(* Logix 5000 project; controller RSL5k_18_Template_noLib Emulate 5570 rev 32.11; software revision 32.02; part 13 of 16 *)
(* tags used below, declared in another part *)
   Ref_FaultCodeList : P_DescList[1];   // Tag containing List of Fault Codes (DINT) and their Descriptions (STRING)
   Inp_LastFaultCode : DINT;   // Most recent drive fault code (enumeration)
   Inp_Ready : BOOL;   // 1=Drive is ready to run
   Inp_Running : BOOL;   // 1=Drive is Running (active)
   Inp_CommandDir : BOOL;   // 1=Drive is commanded Forward, 0=Drive is commanded Reverse
   Inp_Faulted : BOOL;   // 1=Drive has Faulted (see drive display or manual)
   Inp_FwdPermOK : BOOL;   // 1=Permissives OK, drive can start Forward
   Inp_FwdNBPermOK : BOOL;   // 1=Non-Bypassable Permissives OK, drive can start Forward
   Inp_RevPermOK : BOOL;   // 1=Permissives OK, drive can start Reverse
   Inp_RevNBPermOK : BOOL;   // 1=Non-Bypassable Permissives OK, motor can start Reverse
   Inp_IntlkOK : BOOL;   // 1=Interlocks OK, drive can start/run
   Inp_NBIntlkOK : BOOL;   // 1=Non-Bypassable Interlocks OK, drive can start/run
   Inp_IntlkAvail : BOOL;   // 1 = Interlock Availibility OK
   Inp_IOFault : BOOL;   // Input Communication Status 0=OK, 1=fail
   Inp_Sim : BOOL;   // 1=Simulate working drive; 0=Start/Stop/ Monitor actual drive
   Inp_OvrdCmd : DINT;   // Override Command: 0=None, 1=Stop, 2=Start Fwd 3=Start Rev
   Cfg_HasReverse : BOOL;   // 1=Drive can be run reverse, 0=Forward only
   Cfg_HasJog : BOOL;   // 1=Drive Jog Command enabled/visible, 0=Drive Jog Command not allowed
   Cfg_AllowLocal : BOOL;   // 1=Allow Local Start/Stop without alarm, 0=Start/Stop from HMI/prog only
   Cfg_HasRunFdbk : BOOL;   // 1=Drive provides feedback signal on Inp_Running when running
   Cfg_UseRunFdbk : BOOL;   // 1=Drive run feedback should be used for failure checking
   Cfg_HasSpeedFdbk : BOOL;   // 1=Drive provides speed feedback on Inp_SpeedFdbk
   Cfg_HasOutDatalink : BOOL;   // 1=A signal is connected to Out_Datalink
   Cfg_SetTrack : BOOL;   // 1=Settings track for unselected sources, 0=no tracking
   Cfg_SetTrackOvrdHand : BOOL;   // 1=Prog/Oper/Ext Settings track Override/Hand
   Cfg_OperStopPrio : BOOL;   // 1=OCmd_Stop any time, 0=OCmd_Stop only when Oper selected
   Cfg_ExtStopPrio : BOOL;   // 1=XCmd_Stop any time, 0=XCmd_Stop only when Ext selected
   Cfg_OCmdResets : BOOL;   // 1=New drive OCmd resets shed latches and cleared alarms, 0=OCmdReset req'd.
   Cfg_ShedOnFailToStart : BOOL;   // 1=Stop Motor and Alarm on Fail to Start; 0=Alarm only on Fail to Start
   Cfg_ShedOnIOFault : BOOL;   // 1=Stop Motor and Alarm on I/O Fault; 0=Alarm only on I/O Fault
   Cfg_MinSpdRef : REAL;   // Minimum Speed Reference in EU (for limiting)
   Cfg_MaxSpdRef : REAL;   // Maximum Speed Reference in EU (for limiting)
   Cfg_SpeedRefRawMin : REAL;   // Speed Reference Minimum in Drive (raw) Units (for scaling)
   Cfg_SpeedRefRawMax : REAL;   // Speed Reference Maximum in Drive (raw) Units (for scaling)
   Cfg_SpeedRefEUMin : REAL;   // Speed Reference Minimum in Engineering Units (for scaling)
   Cfg_SpeedRefEUMax : REAL;   // Speed Reference Maximum in Engineering Units (for scaling)
   Cfg_OutDatalinkRawMin : REAL;   // Output Datalink Minimum in Drive (raw) Units (for scaling)
   Cfg_OutDatalinkRawMax : REAL;   // Output Datalink Maximum in Drive (raw) Units (for scaling)
   Cfg_OutDatalinkEUMin : REAL;   // Output Datalink Minimum in Engineering Units (for scaling)
   Cfg_OutDatalinkEUMax : REAL;   // Output Datalink Maximum in Engineering Units (for scaling)
   PSet_SpeedRef : REAL;   // Program Setting of Speed Reference (EU)
   PSet_OutDatalink : REAL;   // Program Setting of Output Datalink (EU)
   XSet_SpeedRef : REAL;   // External Setting of Speed Reference (EU)
   XSet_OutDatalink : REAL;   // External Setting of Output Datalink (EU)
   PCmd_StartFwd : BOOL;   // Program Command to Start Drive Forward
   PCmd_StartRev : BOOL;   // Program Command to Start Drive Reverse
   PCmd_Stop : BOOL;   // Program Command to Stop Drive
   PCmd_Reset : BOOL;   // Program Command to Reset drive fault and all Alarms requiring Reset
   XCmd_StartFwd : BOOL;   // External Command to Start Drive Forward
   XCmd_StartRev : BOOL;   // External Command to Start Drive Reverse
   XCmd_Stop : BOOL;   // External Command to Stop Drive
   XCmd_JogFwd : BOOL;   // External Command to Jog Drive Forward
   XCmd_JogRev : BOOL;   // External Command to Jog Drive Reverse
   Out_SpeedRef : REAL;   // Drive Speed Reference in Drive Units (typ. 0-32767 = 0 to max freq.)
   Out_Datalink : REAL;   // Auxiliary Signal (datalink) Output in Drive (raw) Units
   Out_Run : BOOL;   // 1=Start/Run Drive, 0=Stop Drive (for held starter type)
   Out_Stop : BOOL;   // 1=Stop Drive, 0=drive left in current state
   Out_Start : BOOL;   // 1=Start Drive, 0=drive left in current state
   Out_Jog : BOOL;   // 1=Jog drive at Jog Speed, -->0=stop jogging
   Out_ClearFault : BOOL;   // 1=Attempt to clear Drive Fault
   Out_Fwd : BOOL;   // 1=Set drive direction to Forward
   Out_Rev : BOOL;   // 1=Set drive direction to Reverse
   Out_Horn : BOOL;   // 1=Sound audible prior to commanded motor start
   Val_SpeedRef : REAL;   // Speed Reference (target) to drive
   Val_OutDatalink : REAL;   // Output Datalink value to drive
   Val_LastFaultCode : DINT;   // Most recent drive fault code (enumeration)
   Val_Cmd : DINT;   // Device Command 0=None, 1=Stop, 2=StartFwd 3=StartRev 4=JogFwd 5=JogRev
   Sts_Stopped : BOOL;   // 1=Drive requested to stop and is confirmed stopped
   Sts_StartingFwd : BOOL;   // 1=Drive requested to run forward and awaiting run feedback
   Sts_StartingRev : BOOL;   // 1=Drive requested to run reverse and awaiting run feedback
   Sts_RunningFwd : BOOL;   // 1=Drive requested to run and is confirmed running forward
   Sts_RunningRev : BOOL;   // 1=Drive requested to run and is confirmed running reverse
   Sts_StoppingFwd : BOOL;   // 1=Drive running forward requested to stop and awaiting stopped feedback
   Sts_StoppingRev : BOOL;   // 1=Drive running reverse requested to stop and awaiting stopped feedback
   Sts_JoggingFwd : BOOL;   // 1=Drive requested to Jog Forward
   Sts_JoggingRev : BOOL;   // 1=Drive requested to Jog Reverse
   Sts_Horn : BOOL;   // 1=Motor Horn Active
   Sts_CommandDir : BOOL;   // 1=Drive commanded to Forward, 0=Reverse
   Sts_ActualDir : BOOL;   // 1=Drive Actual direction is Forward, 0=Reverse
   Sts_SpeedLimited : BOOL;   // 1=Speed Reference Setting exceeds configured Max/Min limit
   Sts_Available : BOOL;   // 1=Drive available for control by automation (Prog)
   Sts_BypActive : BOOL;   // 1=Bypassing Active (Bypassed or Maintenance)
   Sts_NotRdy : BOOL;   // 1=Device Not Ready, see detail bits for reason
   Nrdy_CfgErr : BOOL;   // 1=Device Not Ready: Configuration Error
   Nrdy_DriveNR : BOOL;   // 1=Device Note Ready: Drive Not Ready
   Nrdy_Fail : BOOL;   // 1=Device Not Ready: Device Failure (Shed Requires Reset)
   Nrdy_Intlk : BOOL;   // 1=Device Not Ready: Interlock Not OK
   Nrdy_IOFault : BOOL;   // 1=Device Not Ready: I/O Fault (Shed Requires Reset)
   Nrdy_OoS : BOOL;   // 1=Device Not Ready: Device is Out of Service
   Nrdy_Perm : BOOL;   // 1=Device Not Ready: Permissive Not OK
   Nrdy_PrioStop : BOOL;   // 1=Device Not Ready: Oper/Ext Priority Stop Requires Reset
   Nrdy_Trip : BOOL;   // 1=Device not Ready: Deivce Tripped (Drive Fault)
   Sts_AlmInh : BOOL;   // 1=An Alarm is Shelved, Disabled or Suppressed, display icon
   Err_RefEU : BOOL;   // 1=Error in Config: Speed Ref EU Min = Max
   Err_OutDLEU : BOOL;   // 1=Error in Config: Output Datalink EU Min = Max
   Sts_Hand : ALIAS FOR CmdSrc.Sts_Hand;
   Sts_OoS : ALIAS FOR CmdSrc.Sts_OoS;
   Sts_Maint : ALIAS FOR CmdSrc.Sts_Maint;
   Sts_Ovrd : ALIAS FOR CmdSrc.Sts_Ovrd;
   Sts_Prog : ALIAS FOR CmdSrc.Sts_Prog;
   Sts_Oper : ALIAS FOR CmdSrc.Sts_Oper;
   Sts_FailToStart : ALIAS FOR FailToStart.Inp;   // 1=Drive Failed to Start (One-Shot)
   Sts_FailToStop : ALIAS FOR FailToStop.Inp;   // 1=Drive Failed to Stop
   Sts_IntlkTrip : ALIAS FOR IntlkTrip.Inp;   // 1=Drive was stopped by an Interlock NOT OK (One-Shot)
   Sts_DriveFault : ALIAS FOR DriveFault.Inp;   // 1=Drive Fault (see drive display or manual)
   Sts_IOFault : ALIAS FOR IOFault.Inp;   // I/O Comm Fault Status (0=OK, 1=Bad)
   P_VSD : BOOL;   // Unique Parameter Name for auto - discovery
   CmdSrc : P_CmdSrc;   // Drive Mode Selection
   IOFault : P_Alarm;   // I/O Fault Alarm
   IntlkTrip : P_Alarm;   // Interlock Trip Alarm
   FailToStop : P_Alarm;   // Drive Failed to Stop Alarm
   FailToStart : P_Alarm;   // Drive Failed to Start Alarm
   Wrk_Run : BOOL;   // 1=Drive should be "running", 0=should be "stopped"
   Wrk_StartRetrigT : TIMER;   // Time to pulse start output on start command retrigger (Maint)
   Wrk_StopRetrigT : TIMER;   // Time to pulse stop output on stop command retrigger (Maint)
   Wrk_RunFdbk : BOOL;   // Run Feedback based on mode, simulation, etc. 1=running
   DriveFault : P_Alarm;   // Drive Faulted Alarm
   Wrk_SpeedRef : REAL;   // Working copy of Speed Reference (for limiting)
   Wrk_Rev : BOOL;   // Working (internal) Direction 1=Reverse 0=Forward (default)
   Wrk_Jog : BOOL;   // 1=Jog Drive, 0=Drive not jogging
   Wrk_ResetT : TIMER;   // Reset Output Pulse Timer
   Wrk_OutDatalink : REAL;   // Selected Output Datalink setting
   Wrk_StopT : TIMER;   // Stop Check Timer (for Fail to Stop)
   Wrk_StartT : TIMER;   // Start Check Timer (for Fail to Start)
   Wrk_Cmd : DINT;   // Buffer for building Val_Cmd
   Wrk_Retrigger : BOOL;   // Maint Start issued while running or Stop while stopped
   Wrk_JogT : TIMER;   // Jog Timer
   Wrk_FaultDescFSC : CONTROL;   // FSC control for Fault Code List search
   Val_FaultDesc : STRING_40;   // Description of Drive Fault (given LastFaultCode)
   Wrk_NotRdyONS : BOOL;   // Assert Stop on One-Shot of Sts_NotRdy
   Wrk_NotRdy : BOOL;   // Device Not Ready conditions excluding shed latches
   Wrk_StartInhT : TIMER;   // Local Start Inhibit Timer
   Wrk_StopInhT : TIMER;   // Local Stop Inhibit Timer
   Wrk_Hand : BOOL;   // Perform Hand Mode alignment with actual device state
   Wrk_StartHornT : TIMER;   // Timer for audible alert or start
   Wrk_StartHorn : BOOL;   // 1=Sound audible prior to commanded motor start
   Wrk_RevPermOK : BOOL;   // Reverse Permissives and NB Permissive OK
   Wrk_FwdPermOK : BOOL;   // Forward Permissives and NB Permissive OK
   OCmd_JogRev : BOOL;   // Operator Command to Jog Drive Reverse (not cleared by instruction!)
   OCmd_JogFwd : BOOL;   // Operator Command to Jog Drive Forward (not cleared by instruction!)
   OCmd_Stop : BOOL;   // Operator Command to Stop Drive
   OCmd_StartRev : BOOL;   // Operator Command to Start Drive Reverse
   OCmd_StartFwd : BOOL;   // Operator Command to Start Drive Forward
   OSet_OutDatalink : REAL;   // Operator Setting of Output Datalink (EU)
   OSet_SpeedRef : REAL;   // Operator Setting of Speed Reference (EU)
   ORdy_JogRev : BOOL;   // 1=Ready for OCmd_JogRev (enabled HMI button)
   ORdy_JogFwd : BOOL;   // 1=Ready for OCmd_JogFwd (enables HMI button)
   ORdy_Stop : BOOL;   // 1=Ready for OCmd_Stop (enables HMI button)
   ORdy_StartRev : BOOL;   // 1=Ready for OCmd_StartRev (enables HMI button)
   ORdy_StartFwd : BOOL;   // 1=Ready for OCmd_StartFwd (enables HMI button)
   Wrk_ExtHas1 : BOOL;   // External has Commands
   Wrk_ProgHas1 : BOOL;   // Program has Commands
   Wrk_OperHas1 : BOOL;   // Operator has Commands
(* P_VSD, continued *)

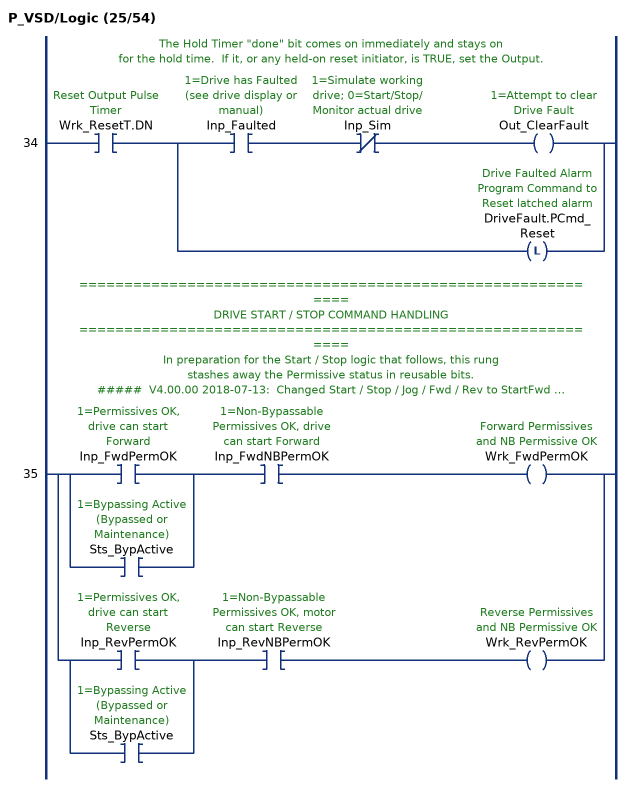
   [picture p277: P_VSD/Logic rungs 34-35]
   // The Hold Timer "done" bit comes on immediately and stays on
   // for the hold time.  If it, or any held-on reset initiator, is TRUE, set the Output.
   34: XIC(Wrk_ResetT.DN)[XIC(Inp_Faulted) XIO(Inp_Sim) OTE(Out_ClearFault) ,OTL(DriveFault.PCmd_Reset) ];
   // ============================================================
   // DRIVE START / STOP COMMAND HANDLING
   // ============================================================
   // In preparation for the Start / Stop logic that follows, this rung
   // stashes away the Permissive status in reusable bits.
   // #####  V4.00.00 2018-07-13:  Changed Start / Stop / Jog / Fwd / Rev to StartFwd / StartRev / Stop / JogFwd / JogRev  #####
   35: [[XIC(Inp_FwdPermOK) ,XIC(Sts_BypActive) ] XIC(Inp_FwdNBPermOK) OTE(Wrk_FwdPermOK) ,[XIC(Inp_RevPermOK) ,XIC(Sts_BypActive) ] XIC(Inp_RevNBPermOK) OTE(Wrk_RevPermOK) ];
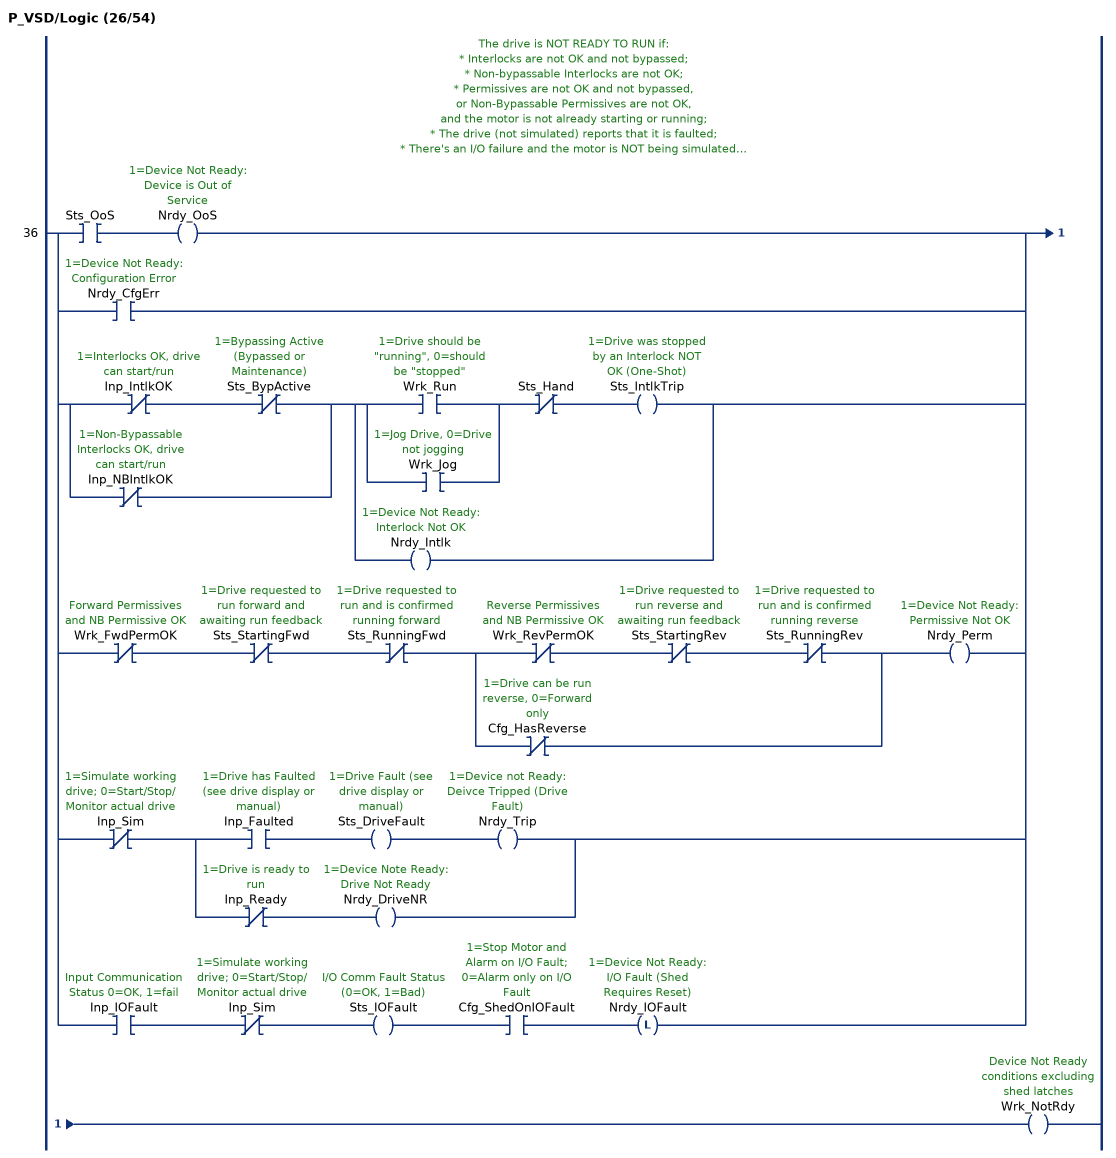
   // The drive is NOT READY TO RUN if:
   // * Interlocks are not OK and not bypassed;
   // * Non-bypassable Interlocks are not OK;
   // * Permissives are not OK and not bypassed,
   // or Non-Bypassable Permissives are not OK,
   // and the motor is not already starting or running;
   // * The drive (not simulated) reports that it is faulted;
   // * There's an I/O failure and the motor is NOT being simulated;
   // * The motor has a Fail to Start that has not been reset;
   // * The drive is disabled (by Maintenance);
   // * This instruction instance has a configuration error.
   // #####  V4.00.00  2018-07-13:  Disable/Enable replaced by P_CmdSrc Out of Service (OoS).  #####
   // #####  V4.00.00  2018-07-13:  Replaced start / stop / fwd / rev with start fwd / start rev / stop  #####
   36: [XIC(Sts_OoS) OTE(Nrdy_OoS) ,XIC(Nrdy_CfgErr) ,[XIO(Inp_IntlkOK) XIO(Sts_BypActive) ,XIO(Inp_NBIntlkOK) ] [[XIC(Wrk_Run) ,XIC(Wrk_Jog) ] XIO(Sts_Hand) OTE(Sts_IntlkTrip) ,OTE(Nrdy_Intlk) ] ,XIO(Wrk_FwdPermOK) XIO(Sts_StartingFwd) XIO(Sts_RunningFwd) [XIO(Wrk_RevPermOK) XIO(Sts_StartingRev) XIO(Sts_RunningRev) ,XIO(Cfg_HasReverse) ] OTE(Nrdy_Perm) ,XIO(Inp_Sim) [XIC(Inp_Faulted) OTE(Sts_DriveFault) OTE(Nrdy_Trip) ,XIO(Inp_Ready) OTE(Nrdy_DriveNR) ] ,XIC(Inp_IOFault) XIO(Inp_Sim) OTE(Sts_IOFault) XIC(Cfg_ShedOnIOFault) OTL(Nrdy_IOFault) ]OTE(Wrk_NotRdy);
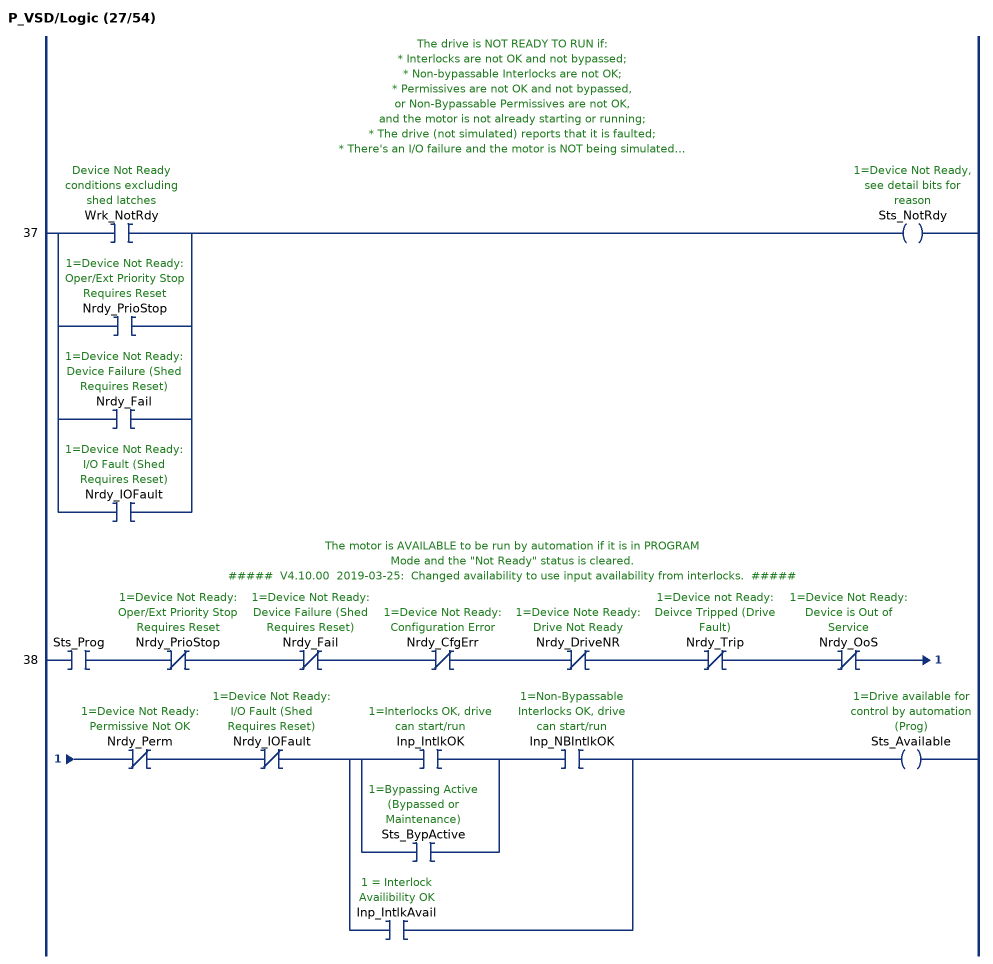
   // The drive is NOT READY TO RUN if:
   // * Interlocks are not OK and not bypassed;
   // * Non-bypassable Interlocks are not OK;
   // * Permissives are not OK and not bypassed,
   // or Non-Bypassable Permissives are not OK,
   // and the motor is not already starting or running;
   // * The drive (not simulated) reports that it is faulted;
   // * There's an I/O failure and the motor is NOT being simulated;
   // * The motor has a Fail to Start that has not been reset;
   // * The drive is disabled (by Maintenance);
   // * This instruction instance has a configuration error.
   37: [XIC(Wrk_NotRdy) ,XIC(Nrdy_PrioStop) ,XIC(Nrdy_Fail) ,XIC(Nrdy_IOFault) ]OTE(Sts_NotRdy);
   // The motor is AVAILABLE to be run by automation if it is in PROGRAM
   // Mode and the "Not Ready" status is cleared.
   // #####  V4.10.00  2019-03-25:  Changed availability to use input availability from interlocks.  #####
   38: XIC(Sts_Prog)XIO(Nrdy_PrioStop)XIO(Nrdy_Fail)XIO(Nrdy_CfgErr)XIO(Nrdy_DriveNR)XIO(Nrdy_Trip)XIO(Nrdy_OoS)XIO(Nrdy_Perm)XIO(Nrdy_IOFault)[[XIC(Inp_IntlkOK) ,XIC(Sts_BypActive) ] XIC(Inp_NBIntlkOK) ,XIC(Inp_IntlkAvail) ]OTE(Sts_Available);
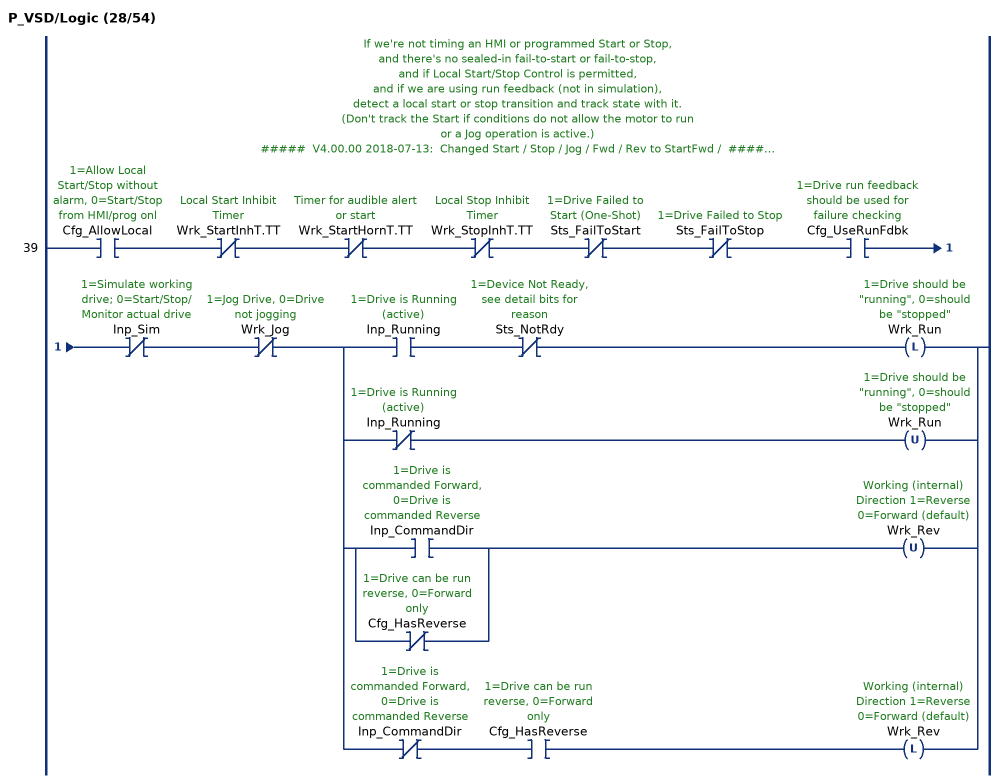
   // If we're not timing an HMI or programmed Start or Stop,
   // and there's no sealed-in fail-to-start or fail-to-stop,
   // and if Local Start/Stop Control is permitted,
   // and if we are using run feedback (not in simulation),
   // detect a local start or stop transition and track state with it.
   // (Don't track the Start if conditions do not allow the motor to run
   // or a Jog operation is active.)
   // #####  V4.00.00 2018-07-13:  Changed Start / Stop / Jog / Fwd / Rev to StartFwd /  #####
   // #####  StartRev / Stop / JogFwd / JogRev.  Deleted Cfg_PCmdClear.  #####
   // ##### V4.00.02  2018-10-30:  Corrected handling Allow Local when horn is enabled.  #####
   39: XIC(Cfg_AllowLocal)XIO(Wrk_StartInhT.TT)XIO(Wrk_StartHornT.TT)XIO(Wrk_StopInhT.TT)XIO(Sts_FailToStart)XIO(Sts_FailToStop)XIC(Cfg_UseRunFdbk)XIO(Inp_Sim)XIO(Wrk_Jog)[XIC(Inp_Running) XIO(Sts_NotRdy) OTL(Wrk_Run) ,XIO(Inp_Running) OTU(Wrk_Run) ,[XIC(Inp_CommandDir) ,XIO(Cfg_HasReverse) ] OTU(Wrk_Rev) ,XIO(Inp_CommandDir) XIC(Cfg_HasReverse) OTL(Wrk_Rev) ];
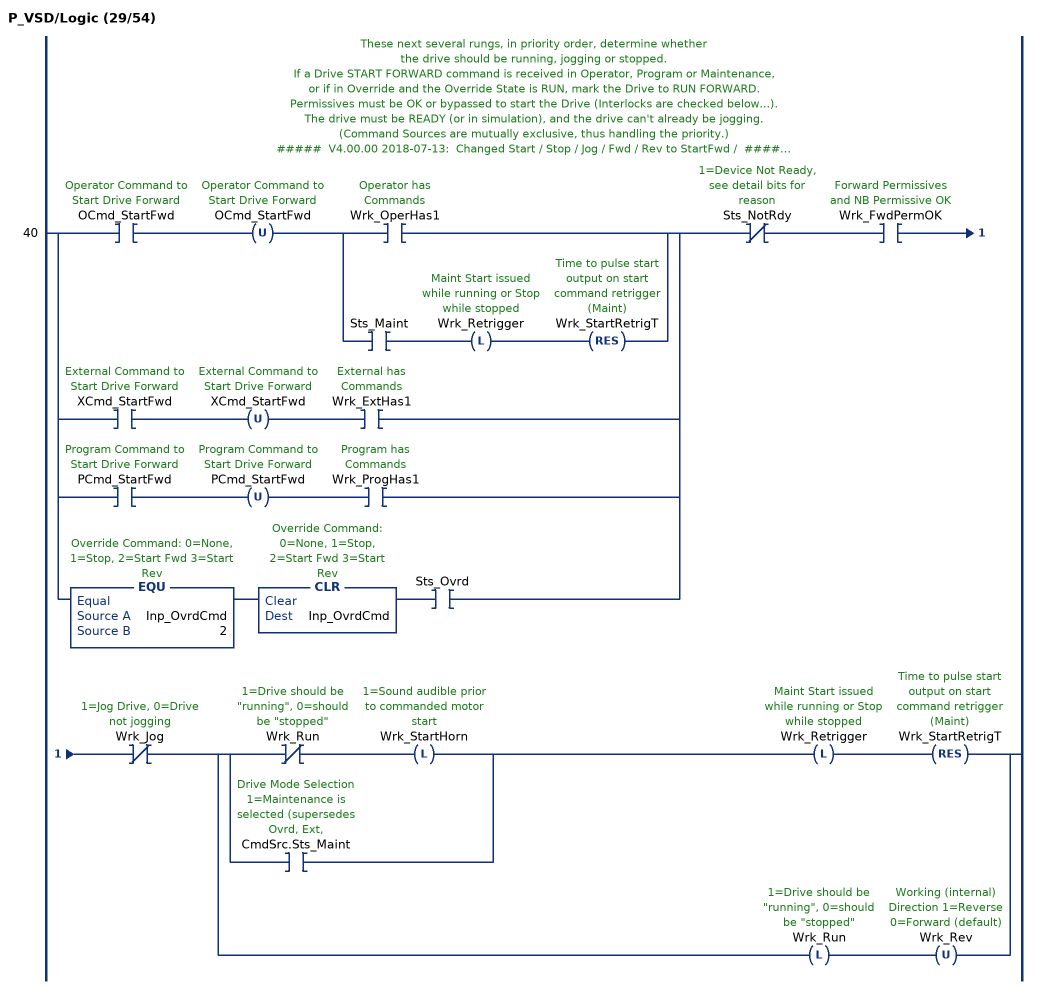
   // These next several rungs, in priority order, determine whether
   // the drive should be running, jogging or stopped.
   // If a Drive START FORWARD command is received in Operator, Program or Maintenance,
   // or if in Override and the Override State is RUN, mark the Drive to RUN FORWARD.
   // Permissives must be OK or bypassed to start the Drive (Interlocks are checked below...).
   // The drive must be READY (or in simulation), and the drive can't already be jogging.
   // (Command Sources are mutually exclusive, thus handling the priority.)
   // #####  V4.00.00 2018-07-13:  Changed Start / Stop / Jog / Fwd / Rev to StartFwd /  #####
   // #####  StartRev / Stop / JogFwd / JogRev.  Deleted Cfg_PCmdClear.  #####
   // #####  Added audible alert prior to commanded start.  #####
   // #####  Changed P_Mode to P_CmdSrc. Added External Command Source and Commands.  #####
   40: [XIC(OCmd_StartFwd) OTU(OCmd_StartFwd) [XIC(Wrk_OperHas1) ,XIC(Sts_Maint) OTL(Wrk_Retrigger) RES(Wrk_StartRetrigT) ] ,XIC(XCmd_StartFwd) OTU(XCmd_StartFwd) XIC(Wrk_ExtHas1) ,XIC(PCmd_StartFwd) OTU(PCmd_StartFwd) XIC(Wrk_ProgHas1) ,EQU(Inp_OvrdCmd,2) CLR(Inp_OvrdCmd) XIC(Sts_Ovrd) ]XIO(Sts_NotRdy)XIC(Wrk_FwdPermOK)XIO(Wrk_Jog)[[XIO(Wrk_Run) OTL(Wrk_StartHorn) ,XIC(CmdSrc.Sts_Maint) ] OTL(Wrk_Retrigger) RES(Wrk_StartRetrigT) ,OTL(Wrk_Run) OTU(Wrk_Rev) ];
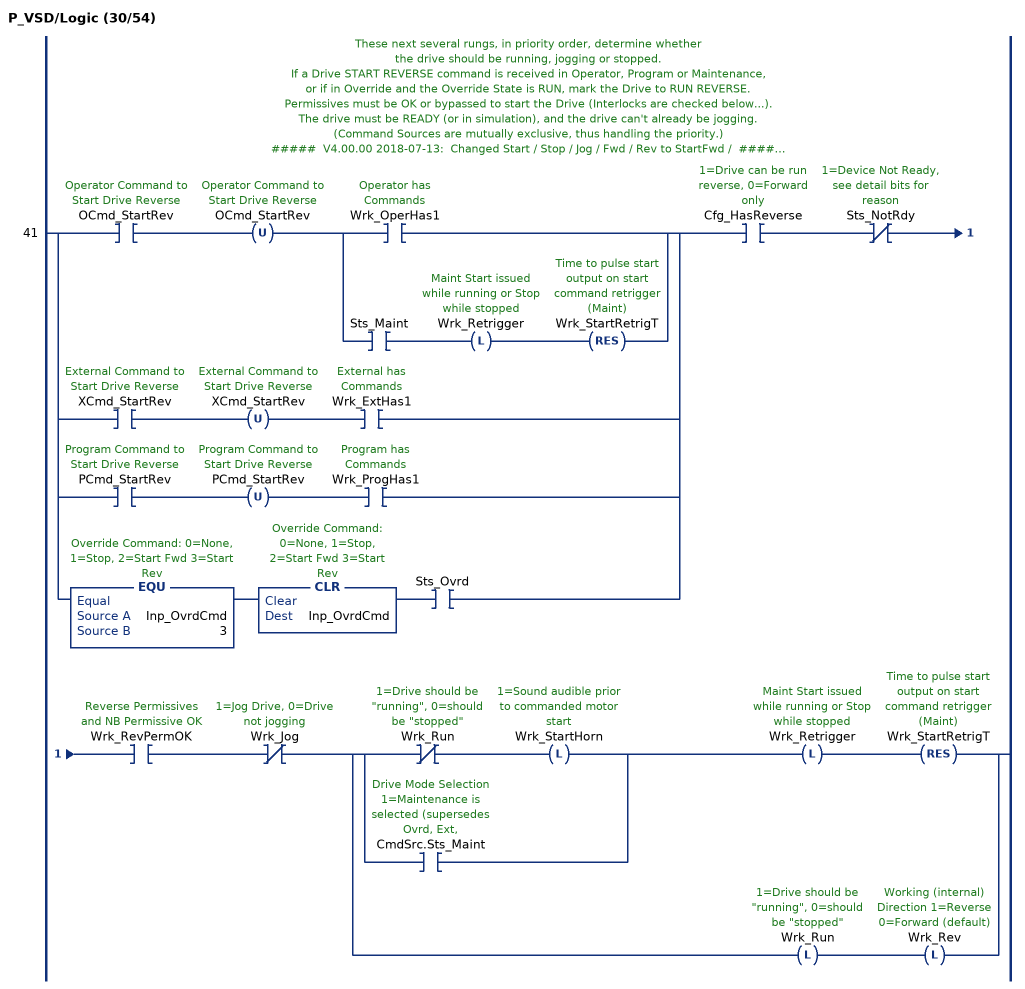
   // These next several rungs, in priority order, determine whether
   // the drive should be running, jogging or stopped.
   // If a Drive START REVERSE command is received in Operator, Program or Maintenance,
   // or if in Override and the Override State is RUN, mark the Drive to RUN REVERSE.
   // Permissives must be OK or bypassed to start the Drive (Interlocks are checked below...).
   // The drive must be READY (or in simulation), and the drive can't already be jogging.
   // (Command Sources are mutually exclusive, thus handling the priority.)
   // #####  V4.00.00 2018-07-13:  Changed Start / Stop / Jog / Fwd / Rev to StartFwd /  #####
   // #####  StartRev / Stop / JogFwd / JogRev.  Deleted Cfg_PCmdClear.  #####
   // #####  Added audible alert prior to commanded start.  #####
   // #####  Changed P_Mode to P_CmdSrc. Added External Command Source and Commands.  #####
   41: [XIC(OCmd_StartRev) OTU(OCmd_StartRev) [XIC(Wrk_OperHas1) ,XIC(Sts_Maint) OTL(Wrk_Retrigger) RES(Wrk_StartRetrigT) ] ,XIC(XCmd_StartRev) OTU(XCmd_StartRev) XIC(Wrk_ExtHas1) ,XIC(PCmd_StartRev) OTU(PCmd_StartRev) XIC(Wrk_ProgHas1) ,EQU(Inp_OvrdCmd,3) CLR(Inp_OvrdCmd) XIC(Sts_Ovrd) ]XIC(Cfg_HasReverse)XIO(Sts_NotRdy)XIC(Wrk_RevPermOK)XIO(Wrk_Jog)[[XIO(Wrk_Run) OTL(Wrk_StartHorn) ,XIC(CmdSrc.Sts_Maint) ] OTL(Wrk_Retrigger) RES(Wrk_StartRetrigT) ,OTL(Wrk_Run) OTL(Wrk_Rev) ];
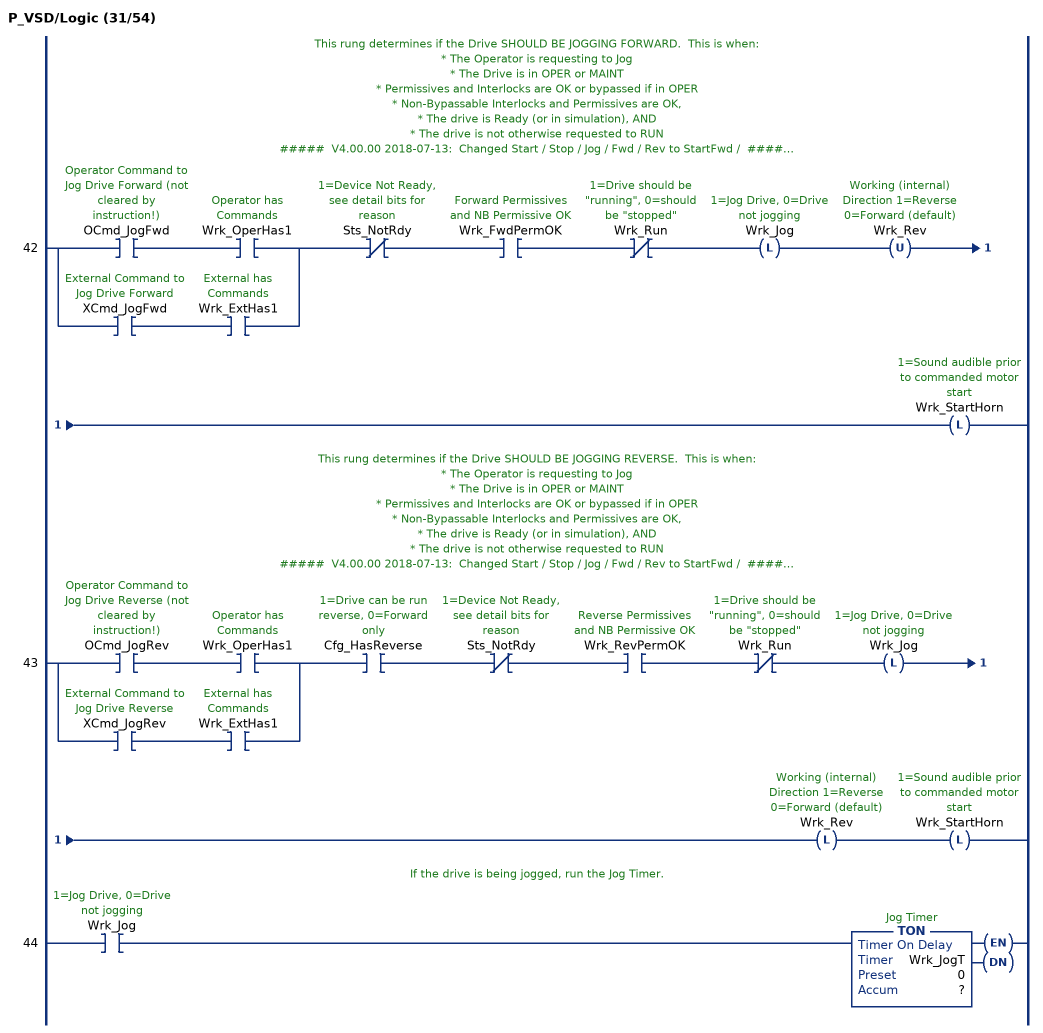
   // This rung determines if the Drive SHOULD BE JOGGING FORWARD.  This is when:
   // * The Operator is requesting to Jog
   // * The Drive is in OPER or MAINT
   // * Permissives and Interlocks are OK or bypassed if in OPER
   // * Non-Bypassable Interlocks and Permissives are OK,
   // * The drive is Ready (or in simulation), AND
   // * The drive is not otherwise requested to RUN
   // #####  V4.00.00 2018-07-13:  Changed Start / Stop / Jog / Fwd / Rev to StartFwd /  #####
   // #####  StartRev / Stop / JogFwd / JogRev.  Deleted Cfg_PCmdClear.  #####
   // #####  Changed P_Mode to P_CmdSrc. Added External Command Source and Commands.  #####
   42: [XIC(OCmd_JogFwd) XIC(Wrk_OperHas1) ,XIC(XCmd_JogFwd) XIC(Wrk_ExtHas1) ]XIO(Sts_NotRdy)XIC(Wrk_FwdPermOK)XIO(Wrk_Run)OTL(Wrk_Jog)OTU(Wrk_Rev)OTL(Wrk_StartHorn);
   // This rung determines if the Drive SHOULD BE JOGGING REVERSE.  This is when:
   // * The Operator is requesting to Jog
   // * The Drive is in OPER or MAINT
   // * Permissives and Interlocks are OK or bypassed if in OPER
   // * Non-Bypassable Interlocks and Permissives are OK,
   // * The drive is Ready (or in simulation), AND
   // * The drive is not otherwise requested to RUN
   // #####  V4.00.00 2018-07-13:  Changed Start / Stop / Jog / Fwd / Rev to StartFwd /  #####
   // #####  StartRev / Stop / JogFwd / JogRev.  Deleted Cfg_PCmdClear.  #####
   // #####  Changed P_Mode to P_CmdSrc. Added External Command Source and Commands.  #####
   43: [XIC(OCmd_JogRev) XIC(Wrk_OperHas1) ,XIC(XCmd_JogRev) XIC(Wrk_ExtHas1) ]XIC(Cfg_HasReverse)XIO(Sts_NotRdy)XIC(Wrk_RevPermOK)XIO(Wrk_Run)OTL(Wrk_Jog)OTL(Wrk_Rev)OTL(Wrk_StartHorn);
   // If the drive is being jogged, run the Jog Timer.
   44: XIC(Wrk_Jog)TON(Wrk_JogT,?,?);
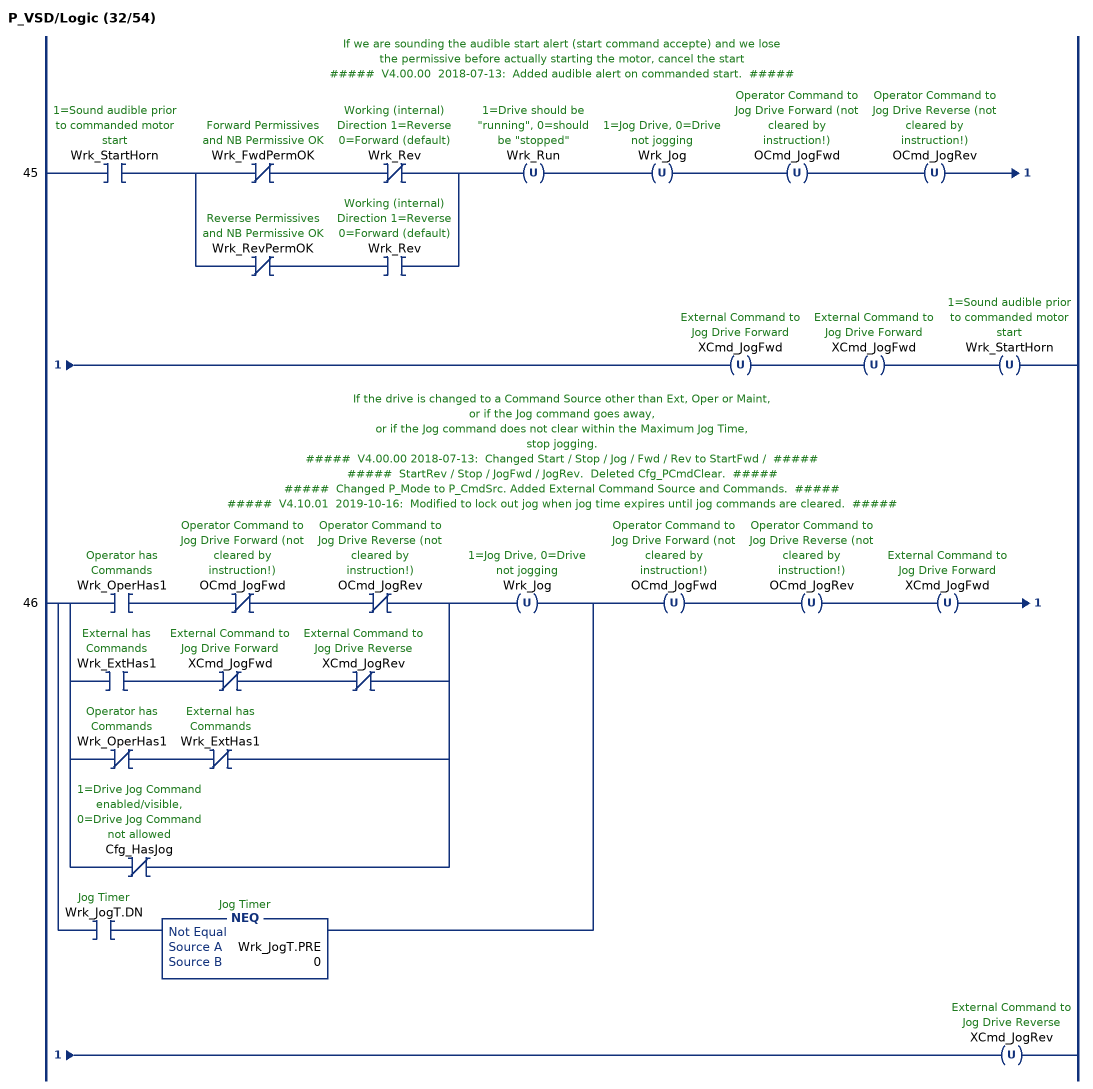
   // If we are sounding the audible start alert (start command accepte) and we lose
   // the permissive before actually starting the motor, cancel the start
   // #####  V4.00.00  2018-07-13:  Added audible alert on commanded start.  #####
   45: XIC(Wrk_StartHorn)[XIO(Wrk_FwdPermOK) XIO(Wrk_Rev) ,XIO(Wrk_RevPermOK) XIC(Wrk_Rev) ]OTU(Wrk_Run)OTU(Wrk_Jog)OTU(OCmd_JogFwd)OTU(OCmd_JogRev)OTU(XCmd_JogFwd)OTU(XCmd_JogFwd)OTU(Wrk_StartHorn);
   // If the drive is changed to a Command Source other than Ext, Oper or Maint,
   // or if the Jog command goes away,
   // or if the Jog command does not clear within the Maximum Jog Time,
   // stop jogging.
   // #####  V4.00.00 2018-07-13:  Changed Start / Stop / Jog / Fwd / Rev to StartFwd /  #####
   // #####  StartRev / Stop / JogFwd / JogRev.  Deleted Cfg_PCmdClear.  #####
   // #####  Changed P_Mode to P_CmdSrc. Added External Command Source and Commands.  #####
   // #####  V4.10.01  2019-10-16:  Modified to lock out jog when jog time expires until jog commands are cleared.  #####
   46: [[XIC(Wrk_OperHas1) XIO(OCmd_JogFwd) XIO(OCmd_JogRev) ,XIC(Wrk_ExtHas1) XIO(XCmd_JogFwd) XIO(XCmd_JogRev) ,XIO(Wrk_OperHas1) XIO(Wrk_ExtHas1) ,XIO(Cfg_HasJog) ] OTU(Wrk_Jog) ,XIC(Wrk_JogT.DN) NEQ(Wrk_JogT.PRE,0) ]OTU(OCmd_JogFwd)OTU(OCmd_JogRev)OTU(XCmd_JogFwd)OTU(XCmd_JogRev);
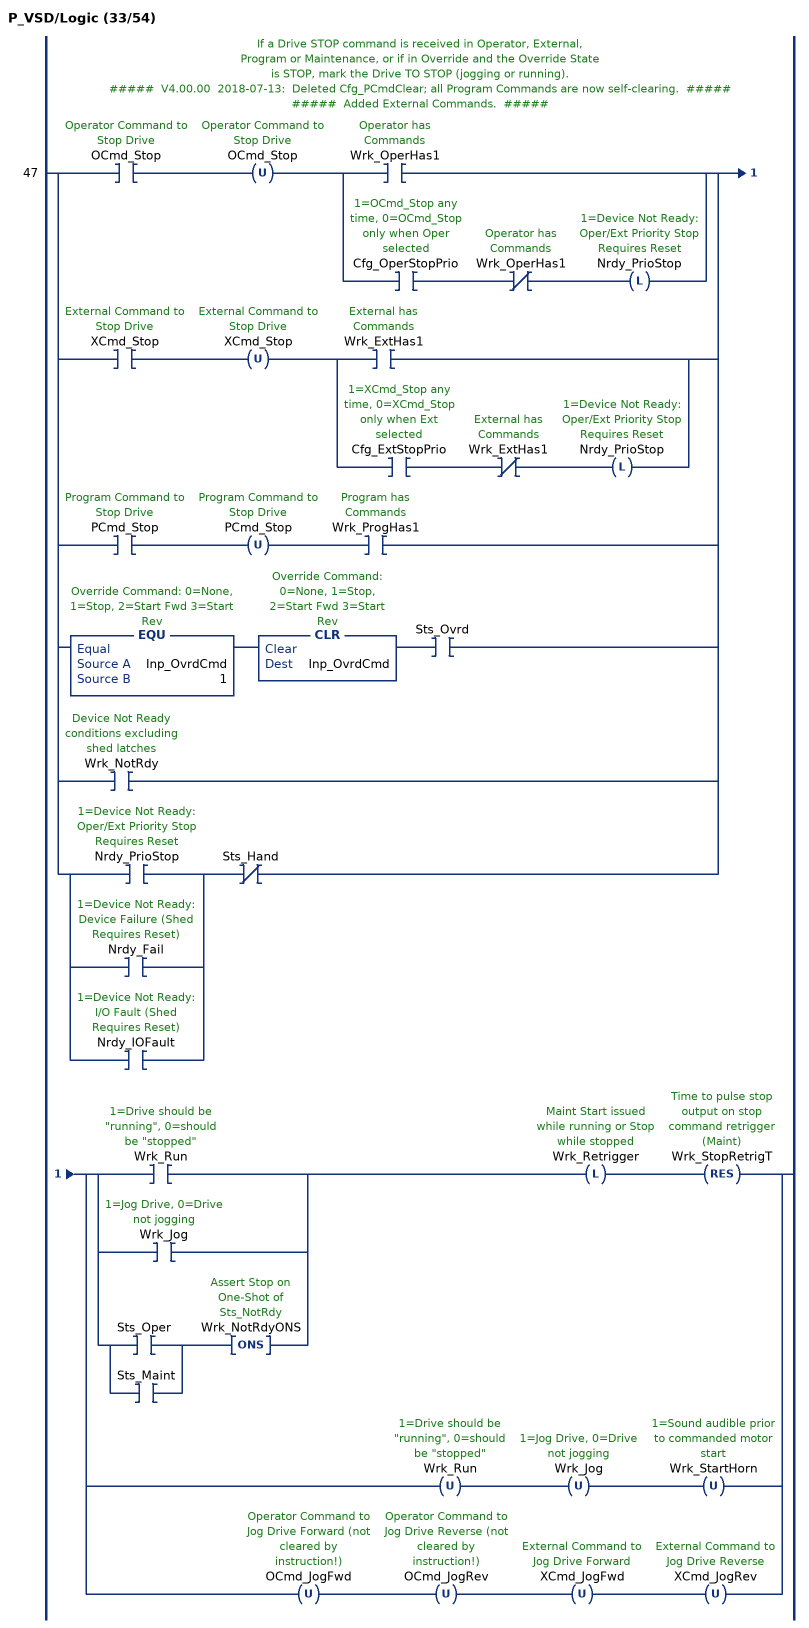
   // If a Drive STOP command is received in Operator, External,
   // Program or Maintenance, or if in Override and the Override State
   // is STOP, mark the Drive TO STOP (jogging or running).
   // #####  V4.00.00  2018-07-13:  Deleted Cfg_PCmdClear; all Program Commands are now self-clearing.  #####
   // #####  Added External Commands.  #####
   47: [XIC(OCmd_Stop) OTU(OCmd_Stop) [XIC(Wrk_OperHas1) ,XIC(Cfg_OperStopPrio) XIO(Wrk_OperHas1) OTL(Nrdy_PrioStop) ] ,XIC(XCmd_Stop) OTU(XCmd_Stop) [XIC(Wrk_ExtHas1) ,XIC(Cfg_ExtStopPrio) XIO(Wrk_ExtHas1) OTL(Nrdy_PrioStop) ] ,XIC(PCmd_Stop) OTU(PCmd_Stop) XIC(Wrk_ProgHas1) ,EQU(Inp_OvrdCmd,1) CLR(Inp_OvrdCmd) XIC(Sts_Ovrd) ,XIC(Wrk_NotRdy) ,[XIC(Nrdy_PrioStop) ,XIC(Nrdy_Fail) ,XIC(Nrdy_IOFault) ] XIO(Sts_Hand) ][[XIC(Wrk_Run) ,XIC(Wrk_Jog) ,[XIC(Sts_Oper) ,XIC(Sts_Maint) ] ONS(Wrk_NotRdyONS) ] OTL(Wrk_Retrigger) RES(Wrk_StopRetrigT) ,OTU(Wrk_Run) OTU(Wrk_Jog) OTU(Wrk_StartHorn) ,OTU(OCmd_JogFwd) OTU(OCmd_JogRev) OTU(XCmd_JogFwd) OTU(XCmd_JogRev) ];
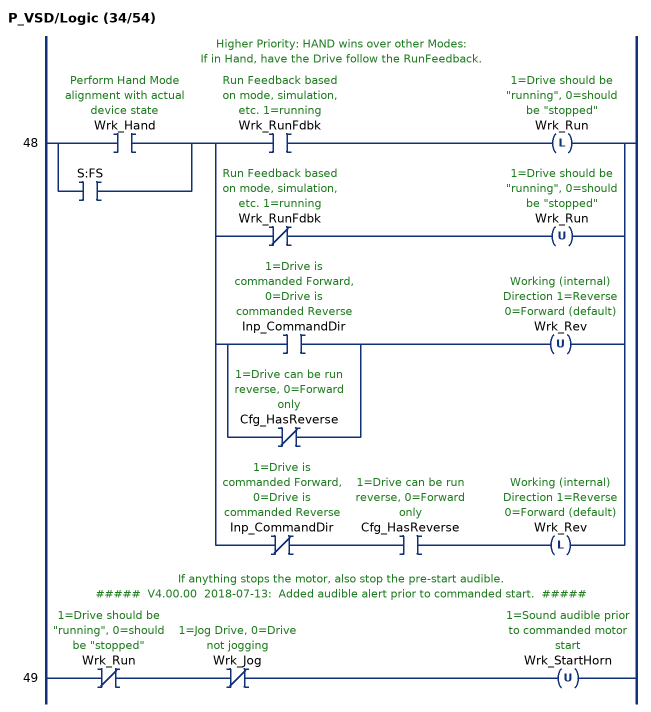
   // Higher Priority: HAND wins over other Modes:
   // If in Hand, have the Drive follow the RunFeedback.
   48: [XIC(Wrk_Hand) ,XIC(S:FS) ][XIC(Wrk_RunFdbk) OTL(Wrk_Run) ,XIO(Wrk_RunFdbk) OTU(Wrk_Run) ,[XIC(Inp_CommandDir) ,XIO(Cfg_HasReverse) ] OTU(Wrk_Rev) ,XIO(Inp_CommandDir) XIC(Cfg_HasReverse) OTL(Wrk_Rev) ];
   // If anything stops the motor, also stop the pre-start audible.
   // #####  V4.00.00  2018-07-13:  Added audible alert prior to commanded start.  #####
   49: XIO(Wrk_Run)XIO(Wrk_Jog)OTU(Wrk_StartHorn);
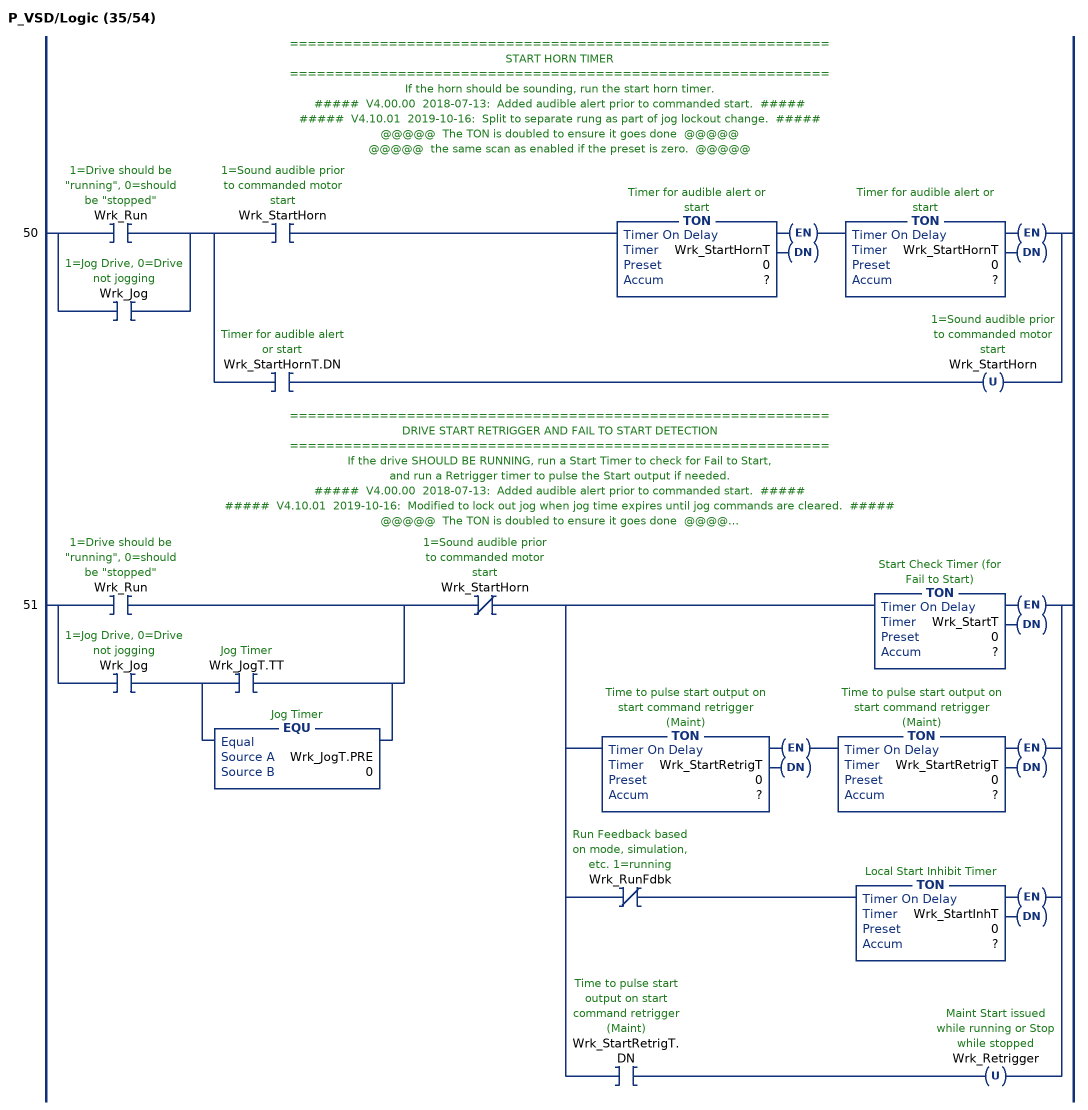
   // ============================================================
   // START HORN TIMER
   // ============================================================
   // If the horn should be sounding, run the start horn timer.
   // #####  V4.00.00  2018-07-13:  Added audible alert prior to commanded start.  #####
   // #####  V4.10.01  2019-10-16:  Split to separate rung as part of jog lockout change.  #####
   // @@@@@  The TON is doubled to ensure it goes done  @@@@@
   // @@@@@  the same scan as enabled if the preset is zero.  @@@@@
   50: [XIC(Wrk_Run) ,XIC(Wrk_Jog) ][XIC(Wrk_StartHorn) TON(Wrk_StartHornT,?,?) TON(Wrk_StartHornT,?,?) ,XIC(Wrk_StartHornT.DN) OTU(Wrk_StartHorn) ];
   // ============================================================
   // DRIVE START RETRIGGER AND FAIL TO START DETECTION
   // ============================================================
   // If the drive SHOULD BE RUNNING, run a Start Timer to check for Fail to Start,
   //  and run a Retrigger timer to pulse the Start output if needed.
   // #####  V4.00.00  2018-07-13:  Added audible alert prior to commanded start.  #####
   // #####  V4.10.01  2019-10-16:  Modified to lock out jog when jog time expires until jog commands are cleared.  #####
   // @@@@@  The TON is doubled to ensure it goes done  @@@@@
   // @@@@@  the same scan as enabled if the preset is zero.  @@@@@
   51: [XIC(Wrk_Run) ,XIC(Wrk_Jog) [XIC(Wrk_JogT.TT) ,EQU(Wrk_JogT.PRE,0) ] ]XIO(Wrk_StartHorn)[TON(Wrk_StartT,?,?) ,TON(Wrk_StartRetrigT,?,?) TON(Wrk_StartRetrigT,?,?) ,XIO(Wrk_RunFdbk) TON(Wrk_StartInhT,?,?) ,XIC(Wrk_StartRetrigT.DN) OTU(Wrk_Retrigger) ];
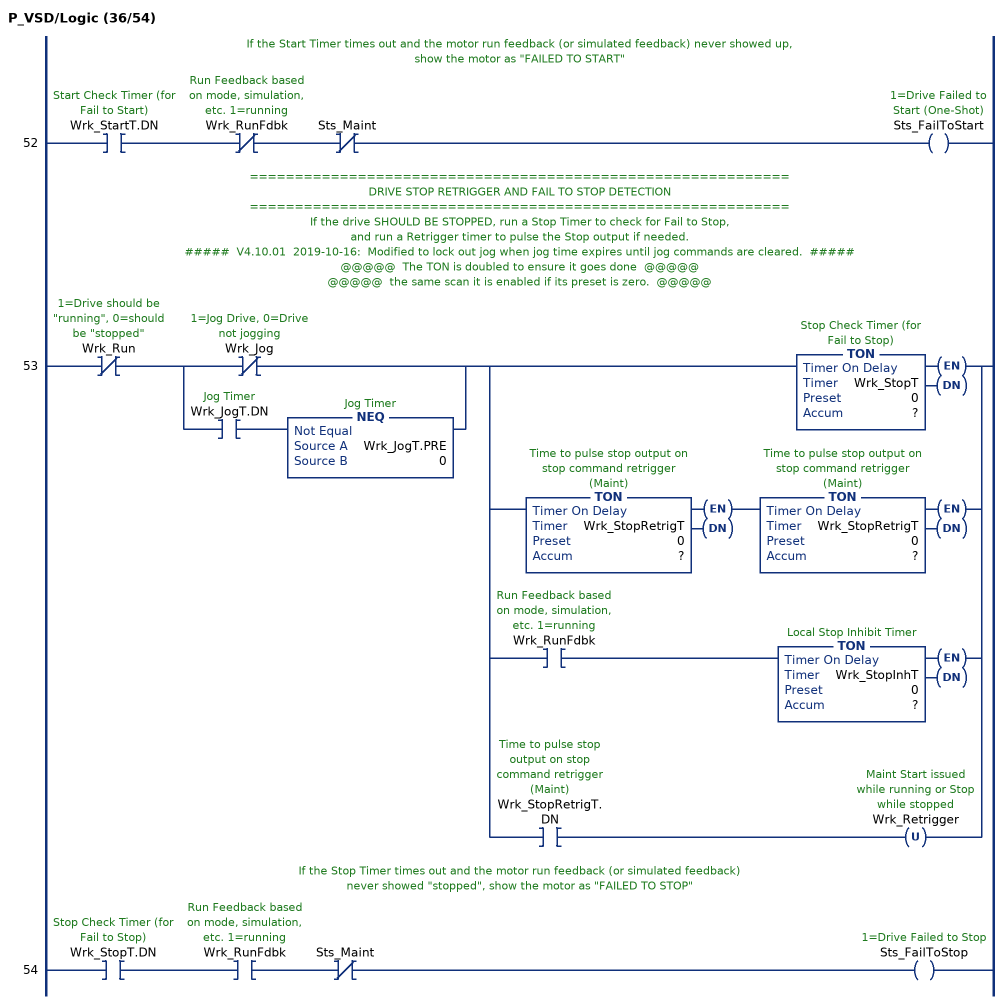
   // If the Start Timer times out and the motor run feedback (or simulated feedback) never showed up,
   // show the motor as "FAILED TO START"
   52: XIC(Wrk_StartT.DN)XIO(Wrk_RunFdbk)XIO(Sts_Maint)OTE(Sts_FailToStart);
   // ============================================================
   // DRIVE STOP RETRIGGER AND FAIL TO STOP DETECTION
   // ============================================================
   // If the drive SHOULD BE STOPPED, run a Stop Timer to check for Fail to Stop,
   //  and run a Retrigger timer to pulse the Stop output if needed.
   // #####  V4.10.01  2019-10-16:  Modified to lock out jog when jog time expires until jog commands are cleared.  #####
   // @@@@@  The TON is doubled to ensure it goes done  @@@@@
   // @@@@@  the same scan it is enabled if its preset is zero.  @@@@@
   53: XIO(Wrk_Run)[XIO(Wrk_Jog) ,XIC(Wrk_JogT.DN) NEQ(Wrk_JogT.PRE,0) ][TON(Wrk_StopT,?,?) ,TON(Wrk_StopRetrigT,?,?) TON(Wrk_StopRetrigT,?,?) ,XIC(Wrk_RunFdbk) TON(Wrk_StopInhT,?,?) ,XIC(Wrk_StopRetrigT.DN) OTU(Wrk_Retrigger) ];
   // If the Stop Timer times out and the motor run feedback (or simulated feedback)
   // never showed "stopped", show the motor as "FAILED TO STOP"
   54: XIC(Wrk_StopT.DN)XIC(Wrk_RunFdbk)XIO(Sts_Maint)OTE(Sts_FailToStop);
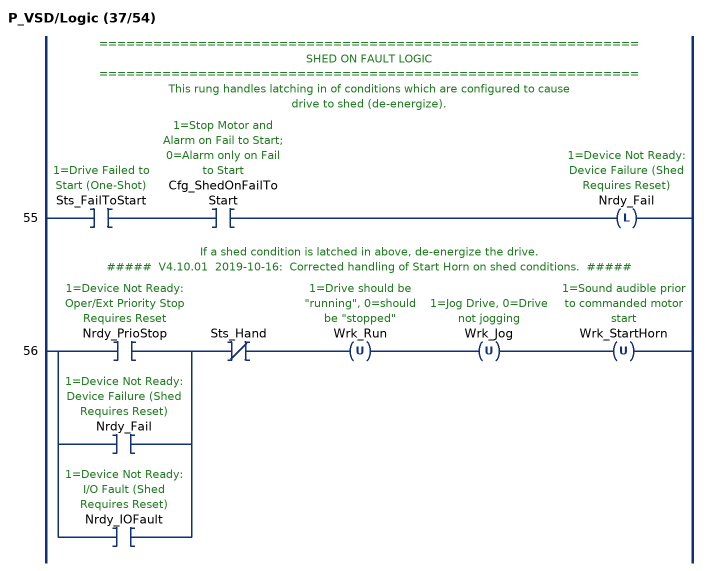
   // ============================================================
   // SHED ON FAULT LOGIC
   // ============================================================
   // This rung handles latching in of conditions which are configured to cause
   // drive to shed (de-energize).
   55: XIC(Sts_FailToStart)XIC(Cfg_ShedOnFailToStart)OTL(Nrdy_Fail);
   // If a shed condition is latched in above, de-energize the drive.
   // #####  V4.10.01  2019-10-16:  Corrected handling of Start Horn on shed conditions.  #####
   56: [XIC(Nrdy_PrioStop) ,XIC(Nrdy_Fail) ,XIC(Nrdy_IOFault) ]XIO(Sts_Hand)OTU(Wrk_Run)OTU(Wrk_Jog)OTU(Wrk_StartHorn);
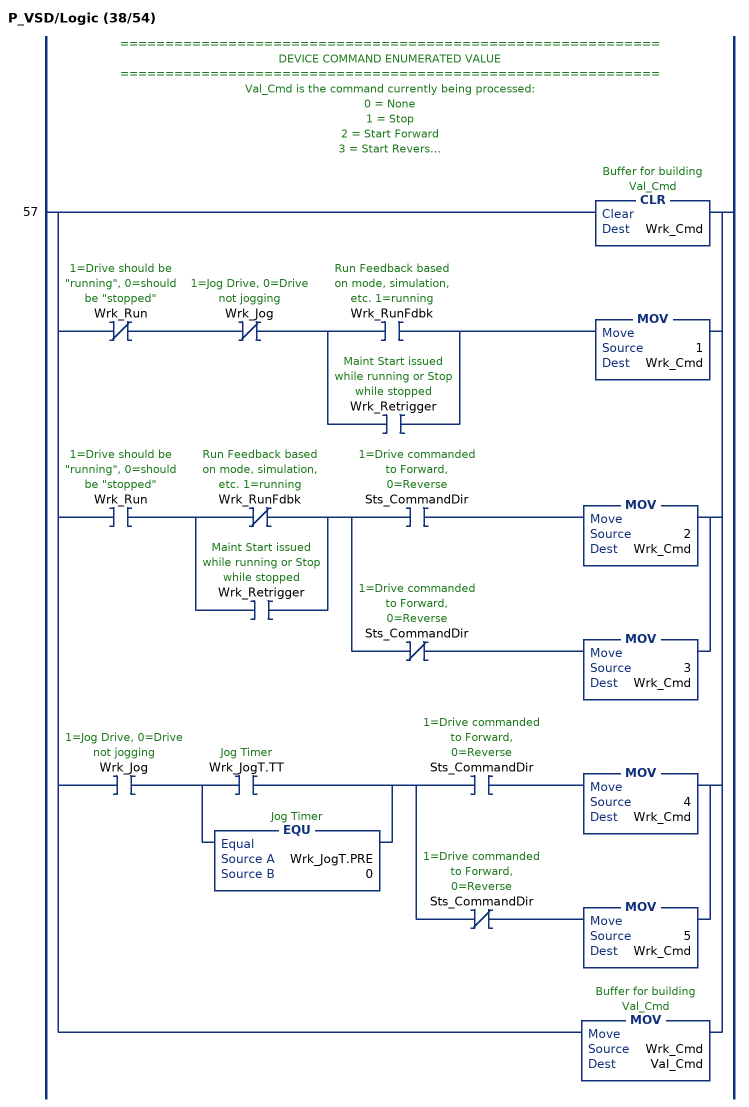
   // ============================================================
   // DEVICE COMMAND ENUMERATED VALUE
   // ============================================================
   // Val_Cmd is the command currently being processed:
   // 0 = None
   // 1 = Stop
   // 2 = Start Forward
   // 3 = Start Reverse
   // 4 = Jog Forward
   // 5 = Jog Reverse
   // #####  V4.10.01  2019-10-16:  Modified to lock out jog when jog time expires until jog commands are cleared.  #####
   57: [CLR(Wrk_Cmd) ,XIO(Wrk_Run) XIO(Wrk_Jog) [XIC(Wrk_RunFdbk) ,XIC(Wrk_Retrigger) ] MOV(1,Wrk_Cmd) ,XIC(Wrk_Run) [XIO(Wrk_RunFdbk) ,XIC(Wrk_Retrigger) ] [XIC(Sts_CommandDir) MOV(2,Wrk_Cmd) ,XIO(Sts_CommandDir) MOV(3,Wrk_Cmd) ] ,XIC(Wrk_Jog) [XIC(Wrk_JogT.TT) ,EQU(Wrk_JogT.PRE,0) ] [XIC(Sts_CommandDir) MOV(4,Wrk_Cmd) ,XIO(Sts_CommandDir) MOV(5,Wrk_Cmd) ] ,MOV(Wrk_Cmd,Val_Cmd) ];
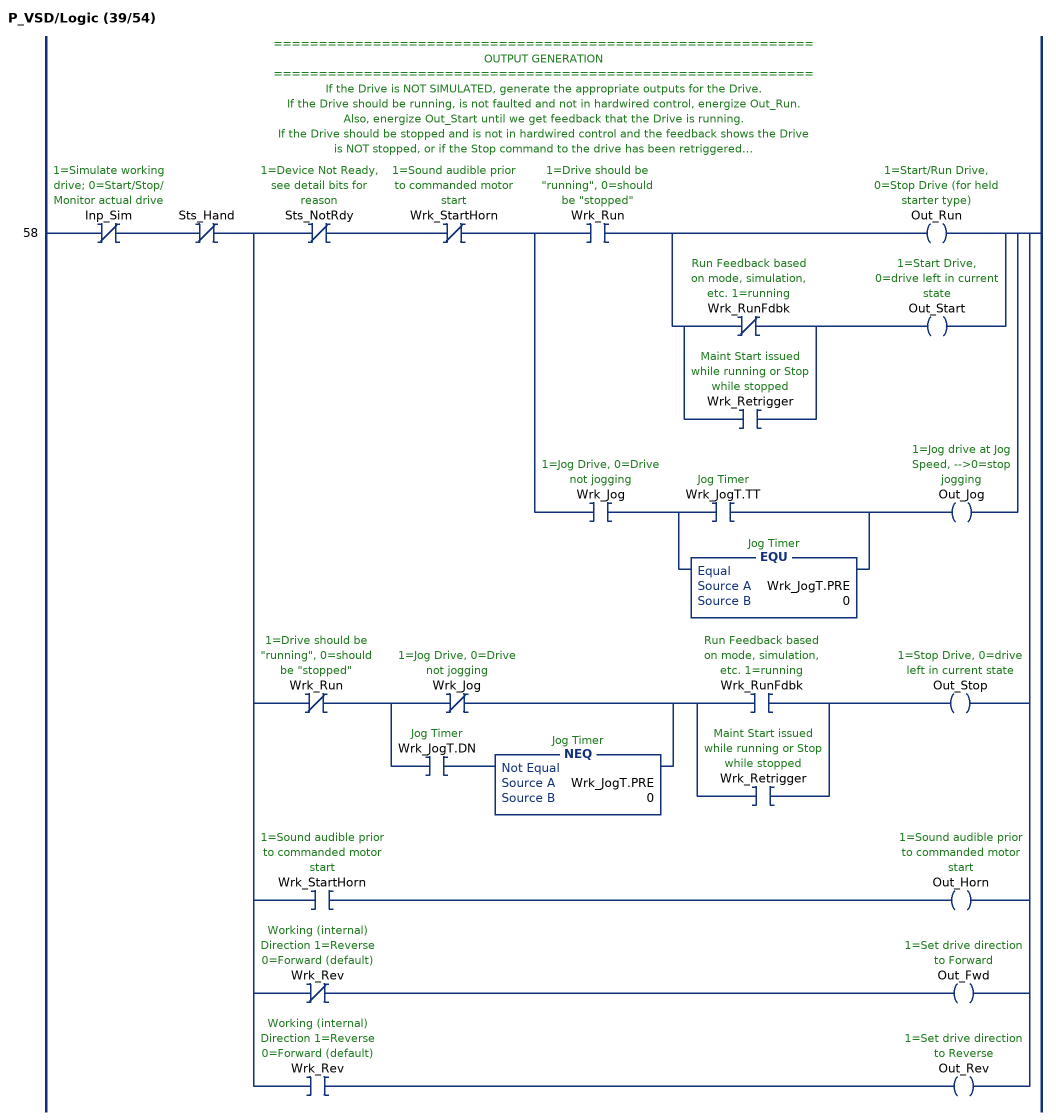
   // ============================================================
   // OUTPUT GENERATION
   // ============================================================
   // If the Drive is NOT SIMULATED, generate the appropriate outputs for the Drive.
   // If the Drive should be running, is not faulted and not in hardwired control, energize Out_Run.
   // Also, energize Out_Start until we get feedback that the Drive is running.
   // If the Drive should be stopped and is not in hardwired control and the feedback shows the Drive
   // is NOT stopped, or if the Stop command to the drive has been retriggered,
   // energize the Out_Stop output to stop the Drive.
   // Finally, if the drive is not simulated, energize the appropriate direction output.
   // #####  V4.00.00  2018-07-13:  Added audible alert prior to commanded start.  #####
   // #####  V4.10.01  2019-10-16:  Modified to lock out jog when jog time expires until jog commands are cleared.  #####
   58: XIO(Inp_Sim)XIO(Sts_Hand)[XIO(Sts_NotRdy) XIO(Wrk_StartHorn) [XIC(Wrk_Run) [OTE(Out_Run) ,[XIO(Wrk_RunFdbk) ,XIC(Wrk_Retrigger) ] OTE(Out_Start) ] ,XIC(Wrk_Jog) [XIC(Wrk_JogT.TT) ,EQU(Wrk_JogT.PRE,0) ] OTE(Out_Jog) ] ,XIO(Wrk_Run) [XIO(Wrk_Jog) ,XIC(Wrk_JogT.DN) NEQ(Wrk_JogT.PRE,0) ] [XIC(Wrk_RunFdbk) ,XIC(Wrk_Retrigger) ] OTE(Out_Stop) ,XIC(Wrk_StartHorn) OTE(Out_Horn) ,XIO(Wrk_Rev) OTE(Out_Fwd) ,XIC(Wrk_Rev) OTE(Out_Rev) ];
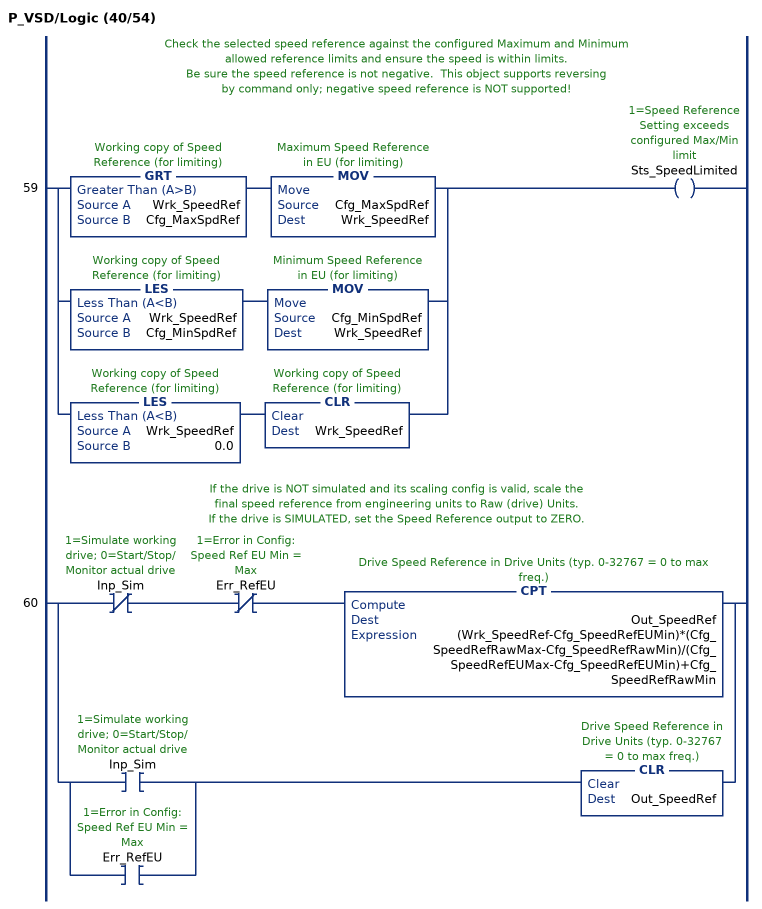
   // Check the selected speed reference against the configured Maximum and Minimum
   // allowed reference limits and ensure the speed is within limits.
   // Be sure the speed reference is not negative.  This object supports reversing
   // by command only; negative speed reference is NOT supported!
   59: [GRT(Wrk_SpeedRef,Cfg_MaxSpdRef) MOV(Cfg_MaxSpdRef,Wrk_SpeedRef) ,LES(Wrk_SpeedRef,Cfg_MinSpdRef) MOV(Cfg_MinSpdRef,Wrk_SpeedRef) ,LES(Wrk_SpeedRef,0.0) CLR(Wrk_SpeedRef) ]OTE(Sts_SpeedLimited);
   // If the drive is NOT simulated and its scaling config is valid, scale the
   // final speed reference from engineering units to Raw (drive) Units.
   // If the drive is SIMULATED, set the Speed Reference output to ZERO.
   60: [XIO(Inp_Sim) XIO(Err_RefEU) CPT(Out_SpeedRef,(Wrk_SpeedRef-Cfg_SpeedRefEUMin)*(Cfg_SpeedRefRawMax-Cfg_SpeedRefRawMin)/(Cfg_SpeedRefEUMax-Cfg_SpeedRefEUMin)+Cfg_SpeedRefRawMin) ,[XIC(Inp_Sim) ,XIC(Err_RefEU) ] CLR(Out_SpeedRef) ];
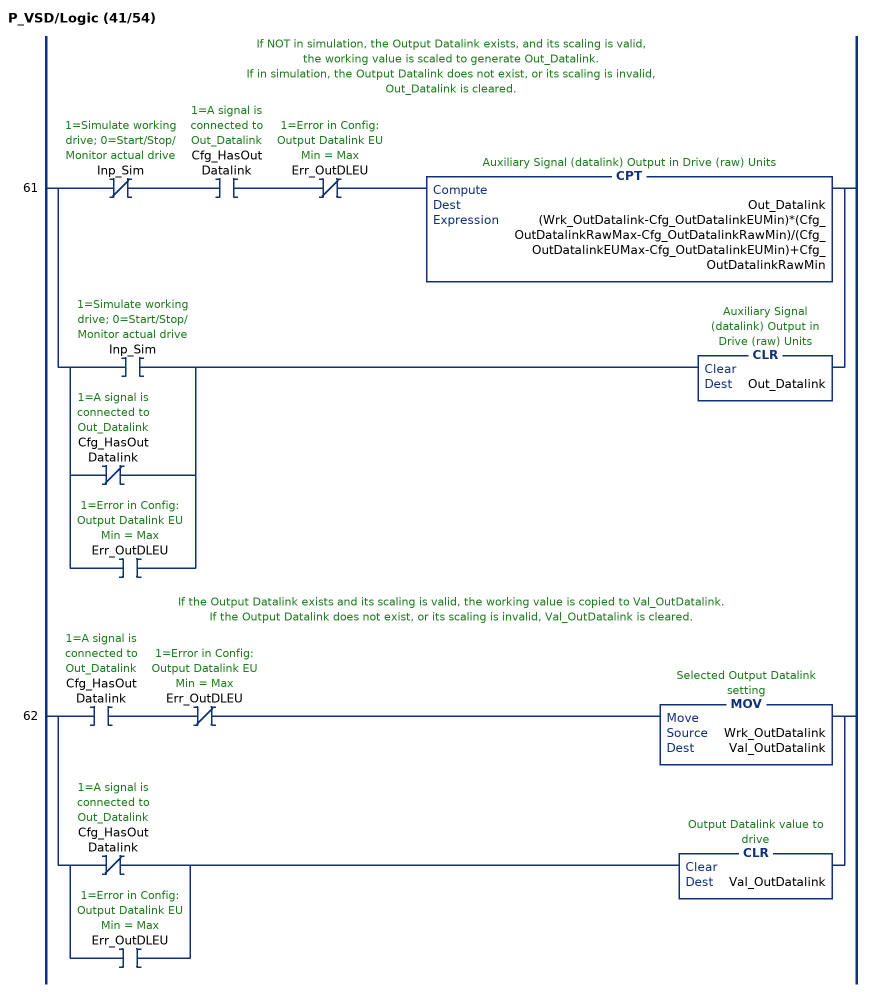
   // If NOT in simulation, the Output Datalink exists, and its scaling is valid,
   // the working value is scaled to generate Out_Datalink.
   // If in simulation, the Output Datalink does not exist, or its scaling is invalid,
   // Out_Datalink is cleared.
   61: [XIO(Inp_Sim) XIC(Cfg_HasOutDatalink) XIO(Err_OutDLEU) CPT(Out_Datalink,(Wrk_OutDatalink-Cfg_OutDatalinkEUMin)*(Cfg_OutDatalinkRawMax-Cfg_OutDatalinkRawMin)/(Cfg_OutDatalinkEUMax-Cfg_OutDatalinkEUMin)+Cfg_OutDatalinkRawMin) ,[XIC(Inp_Sim) ,XIO(Cfg_HasOutDatalink) ,XIC(Err_OutDLEU) ] CLR(Out_Datalink) ];
   // If the Output Datalink exists and its scaling is valid, the working value is copied to Val_OutDatalink.
   // If the Output Datalink does not exist, or its scaling is invalid, Val_OutDatalink is cleared.
   62: [XIC(Cfg_HasOutDatalink) XIO(Err_OutDLEU) MOV(Wrk_OutDatalink,Val_OutDatalink) ,[XIO(Cfg_HasOutDatalink) ,XIC(Err_OutDLEU) ] CLR(Val_OutDatalink) ];
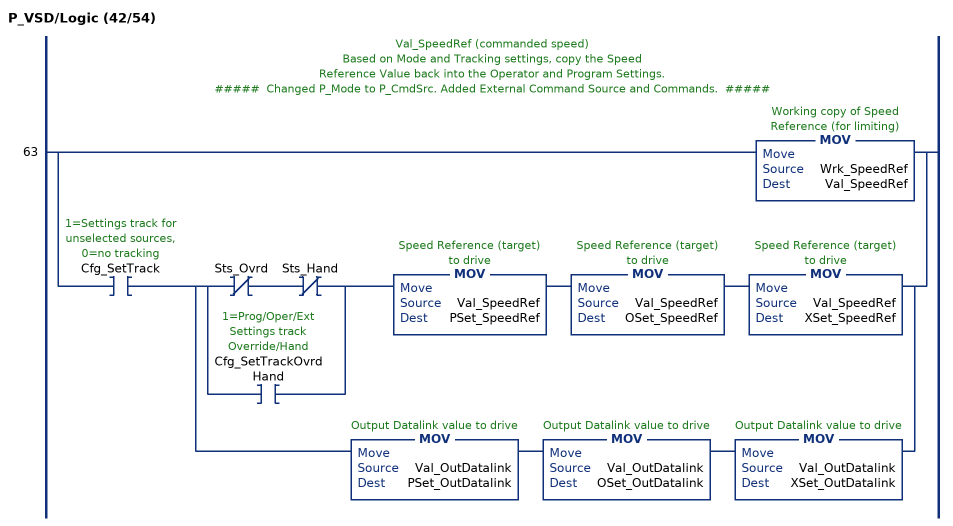
   // Val_SpeedRef (commanded speed)
   // Based on Mode and Tracking settings, copy the Speed
   // Reference Value back into the Operator and Program Settings.
   // #####  Changed P_Mode to P_CmdSrc. Added External Command Source and Commands.  #####
   63: [MOV(Wrk_SpeedRef,Val_SpeedRef) ,XIC(Cfg_SetTrack) [[XIO(Sts_Ovrd) XIO(Sts_Hand) ,XIC(Cfg_SetTrackOvrdHand) ] MOV(Val_SpeedRef,PSet_SpeedRef) MOV(Val_SpeedRef,OSet_SpeedRef) MOV(Val_SpeedRef,XSet_SpeedRef) ,MOV(Val_OutDatalink,PSet_OutDatalink) MOV(Val_OutDatalink,OSet_OutDatalink) MOV(Val_OutDatalink,XSet_OutDatalink) ] ];
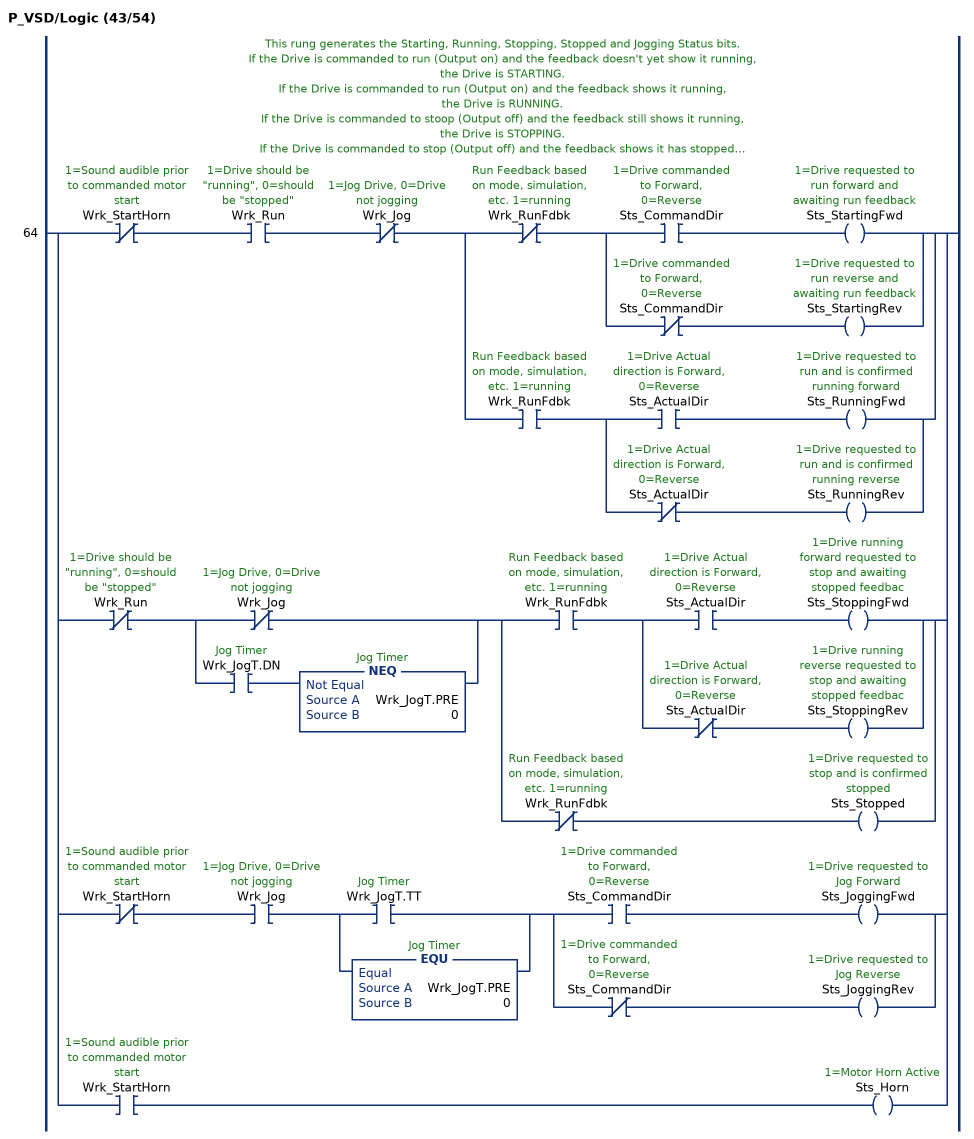
   // This rung generates the Starting, Running, Stopping, Stopped and Jogging Status bits.
   // If the Drive is commanded to run (Output on) and the feedback doesn't yet show it running,
   // the Drive is STARTING.
   // If the Drive is commanded to run (Output on) and the feedback shows it running,
   // the Drive is RUNNING.
   // If the Drive is commanded to stoop (Output off) and the feedback still shows it running,
   // the Drive is STOPPING.
   // If the Drive is commanded to stop (Output off) and the feedback shows it has stopped,
   // the Drive is STOPPED.
   // If the Drive is commanded to jog, show the status as JOGGING.
   // If the audible alert is active, show the Status as HORN.
   // #####  V4.00.00 2018-07-13:  Changed Start / Stop / Jog / Fwd / Rev to StartFwd / StartRev / Stop / JogFwd / JogRev  #####
   // #####  V4.10.00  2019-03-25:  Added Horn Status.  #####
   // #####  V4.10.01  2019-10-16:  Modified to lock out jog when jog time expires until jog commands are cleared.  #####
   64: [XIO(Wrk_StartHorn) XIC(Wrk_Run) XIO(Wrk_Jog) [XIO(Wrk_RunFdbk) [XIC(Sts_CommandDir) OTE(Sts_StartingFwd) ,XIO(Sts_CommandDir) OTE(Sts_StartingRev) ] ,XIC(Wrk_RunFdbk) [XIC(Sts_ActualDir) OTE(Sts_RunningFwd) ,XIO(Sts_ActualDir) OTE(Sts_RunningRev) ] ] ,XIO(Wrk_Run) [XIO(Wrk_Jog) ,XIC(Wrk_JogT.DN) NEQ(Wrk_JogT.PRE,0) ] [XIC(Wrk_RunFdbk) [XIC(Sts_ActualDir) OTE(Sts_StoppingFwd) ,XIO(Sts_ActualDir) OTE(Sts_StoppingRev) ] ,XIO(Wrk_RunFdbk) OTE(Sts_Stopped) ] ,XIO(Wrk_StartHorn) XIC(Wrk_Jog) [XIC(Wrk_JogT.TT) ,EQU(Wrk_JogT.PRE,0) ] [XIC(Sts_CommandDir) OTE(Sts_JoggingFwd) ,XIO(Sts_CommandDir) OTE(Sts_JoggingRev) ] ,XIC(Wrk_StartHorn) OTE(Sts_Horn) ];
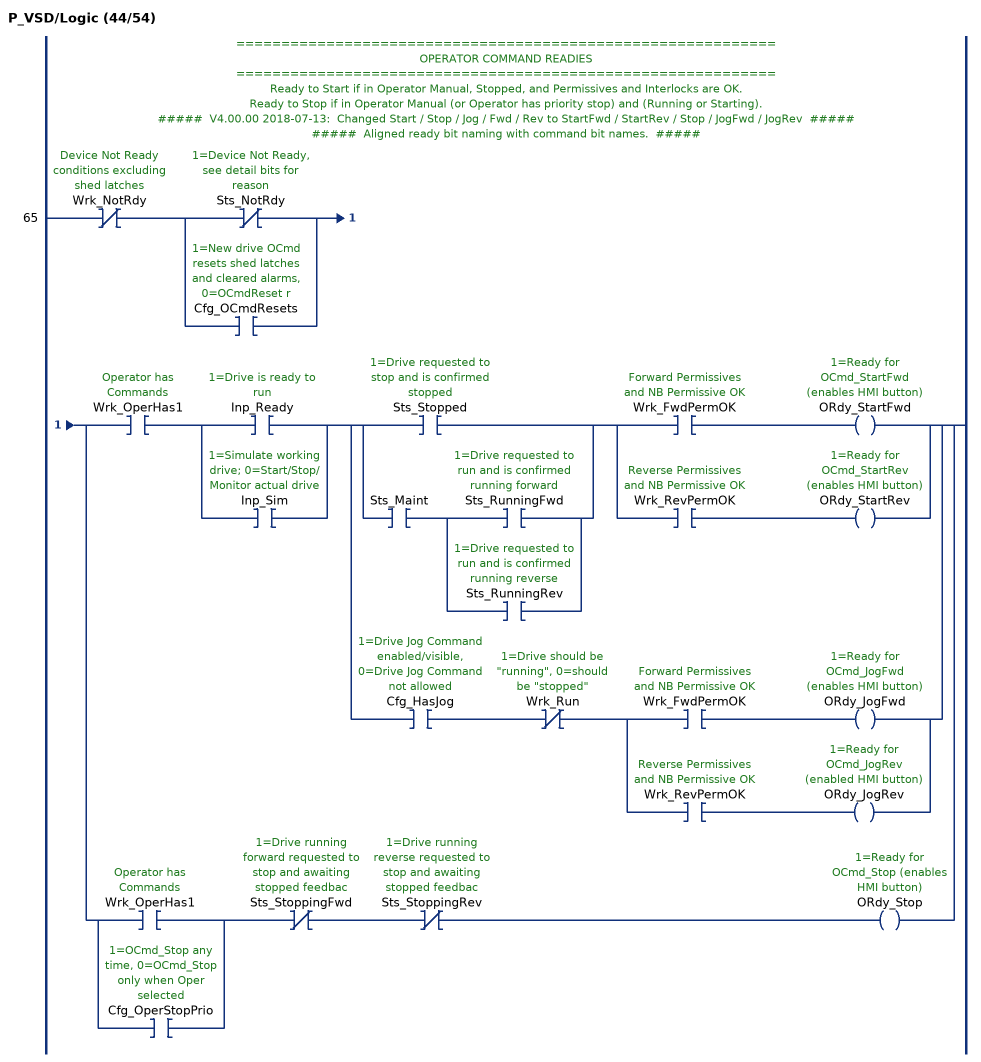
   // ============================================================
   // OPERATOR COMMAND READIES
   // ============================================================
   // Ready to Start if in Operator Manual, Stopped, and Permissives and Interlocks are OK.
   // Ready to Stop if in Operator Manual (or Operator has priority stop) and (Running or Starting).
   // #####  V4.00.00 2018-07-13:  Changed Start / Stop / Jog / Fwd / Rev to StartFwd / StartRev / Stop / JogFwd / JogRev  #####
   // #####  Aligned ready bit naming with command bit names.  #####
   65: XIO(Wrk_NotRdy)[XIO(Sts_NotRdy) ,XIC(Cfg_OCmdResets) ][XIC(Wrk_OperHas1) [XIC(Inp_Ready) ,XIC(Inp_Sim) ] [[XIC(Sts_Stopped) ,XIC(Sts_Maint) [XIC(Sts_RunningFwd) ,XIC(Sts_RunningRev) ] ] [XIC(Wrk_FwdPermOK) OTE(ORdy_StartFwd) ,XIC(Wrk_RevPermOK) OTE(ORdy_StartRev) ] ,XIC(Cfg_HasJog) XIO(Wrk_Run) [XIC(Wrk_FwdPermOK) OTE(ORdy_JogFwd) ,XIC(Wrk_RevPermOK) OTE(ORdy_JogRev) ] ] ,[XIC(Wrk_OperHas1) ,XIC(Cfg_OperStopPrio) ] XIO(Sts_StoppingFwd) XIO(Sts_StoppingRev) OTE(ORdy_Stop) ];
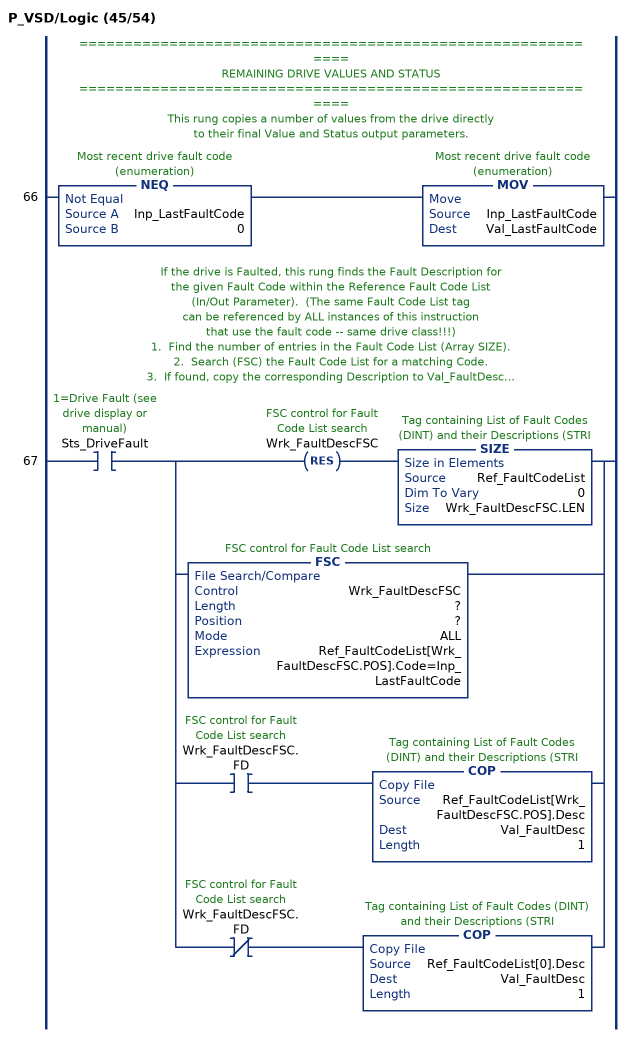
   // ============================================================
   // REMAINING DRIVE VALUES AND STATUS
   // ============================================================
   // This rung copies a number of values from the drive directly
   // to their final Value and Status output parameters.
   66: NEQ(Inp_LastFaultCode,0)MOV(Inp_LastFaultCode,Val_LastFaultCode);
   // If the drive is Faulted, this rung finds the Fault Description for
   // the given Fault Code within the Reference Fault Code List
   // (In/Out Parameter).  (The same Fault Code List tag
   // can be referenced by ALL instances of this instruction
   // that use the fault code -- same drive class!!!)
   // 1.  Find the number of entries in the Fault Code List (Array SIZE).
   // 2.  Search (FSC) the Fault Code List for a matching Code.
   // 3.  If found, copy the corresponding Description to Val_FaultDesc.
   // 4.  If NOT found, copy list entry zero ("No Help Available for this code").
   67: XIC(Sts_DriveFault)[RES(Wrk_FaultDescFSC) SIZE(Ref_FaultCodeList,0,Wrk_FaultDescFSC.LEN) ,FSC(Wrk_FaultDescFSC,?,?,ALL,Ref_FaultCodeList[Wrk_FaultDescFSC.POS].Code=Inp_LastFaultCode) ,XIC(Wrk_FaultDescFSC.FD) COP(Ref_FaultCodeList[Wrk_FaultDescFSC.POS].Desc,Val_FaultDesc,1) ,XIO(Wrk_FaultDescFSC.FD) COP(Ref_FaultCodeList[0].Desc,Val_FaultDesc,1) ];
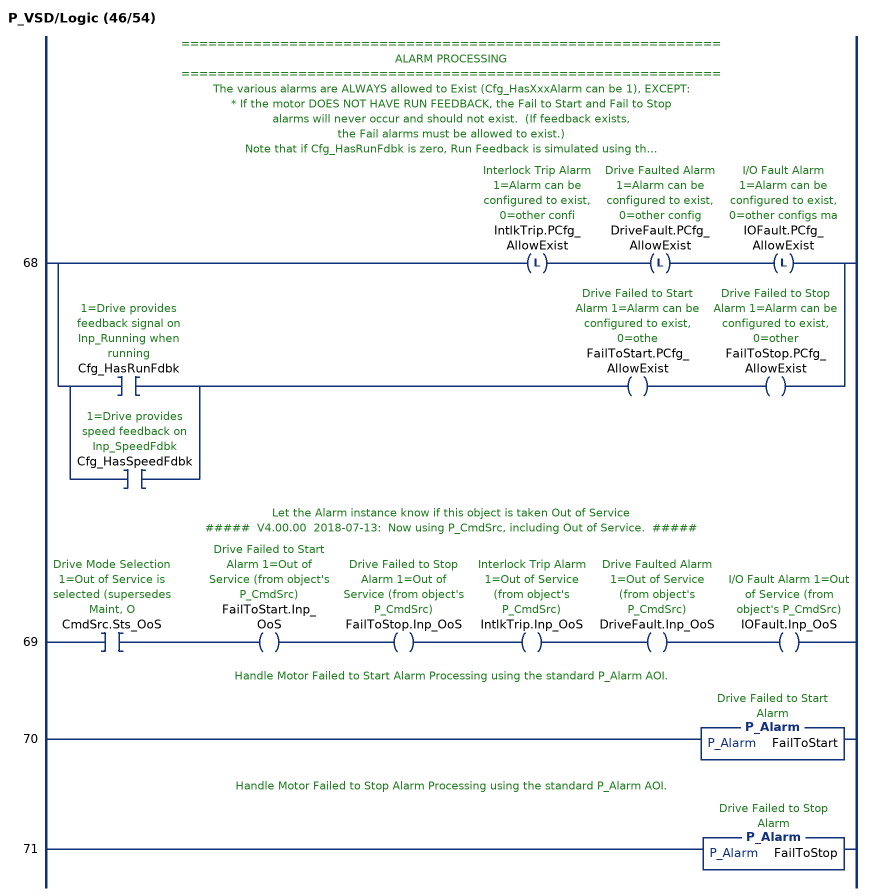
   // ============================================================
   // ALARM PROCESSING
   // ============================================================
   // The various alarms are ALWAYS allowed to Exist (Cfg_HasXxxAlarm can be 1), EXCEPT:
   // * If the motor DOES NOT HAVE RUN FEEDBACK, the Fail to Start and Fail to Stop
   // alarms will never occur and should not exist.  (If feedback exists,
   // the Fail alarms must be allowed to exist.)
   // Note that if Cfg_HasRunFdbk is zero, Run Feedback is simulated using the
   // Speed Feedback, if the drive has that!
   // #####  V4.00.00  2018-07-13:  Deleted Cfg_PCmdClear; all Program Commands are now self-clearing.  #####
   68: [OTL(IntlkTrip.PCfg_AllowExist) OTL(DriveFault.PCfg_AllowExist) OTL(IOFault.PCfg_AllowExist) ,[XIC(Cfg_HasRunFdbk) ,XIC(Cfg_HasSpeedFdbk) ] OTE(FailToStart.PCfg_AllowExist) OTE(FailToStop.PCfg_AllowExist) ];
   // Let the Alarm instance know if this object is taken Out of Service
   // #####  V4.00.00  2018-07-13:  Now using P_CmdSrc, including Out of Service.  #####
   69: XIC(CmdSrc.Sts_OoS)OTE(FailToStart.Inp_OoS)OTE(FailToStop.Inp_OoS)OTE(IntlkTrip.Inp_OoS)OTE(DriveFault.Inp_OoS)OTE(IOFault.Inp_OoS);
   // Handle Motor Failed to Start Alarm Processing using the standard P_Alarm AOI.
   70: P_Alarm(FailToStart);
   // Handle Motor Failed to Stop Alarm Processing using the standard P_Alarm AOI.
   71: P_Alarm(FailToStop);
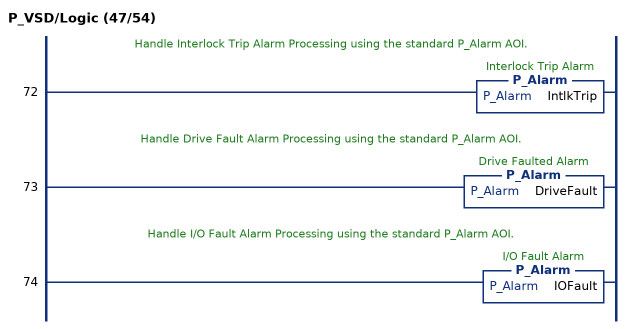
   // Handle Interlock Trip Alarm Processing using the standard P_Alarm AOI.
   72: P_Alarm(IntlkTrip);
   // Handle Drive Fault Alarm Processing using the standard P_Alarm AOI.
   73: P_Alarm(DriveFault);
   // Handle I/O Fault Alarm Processing using the standard P_Alarm AOI.
   74: P_Alarm(IOFault);
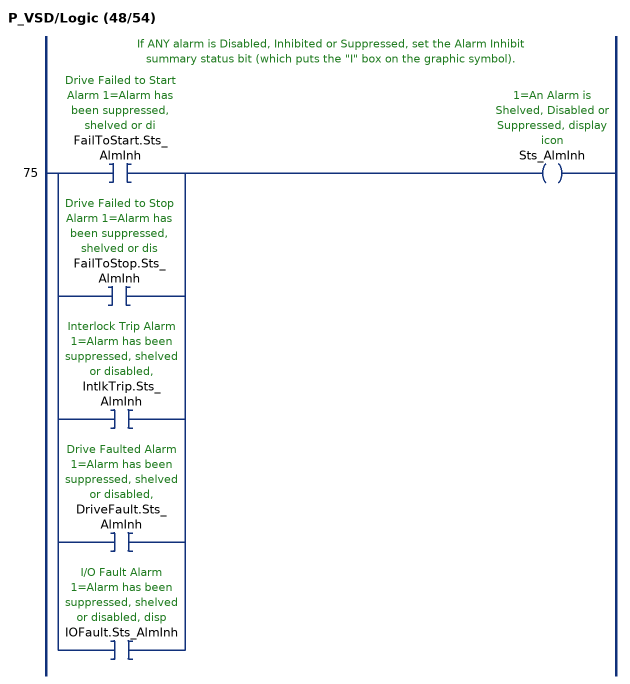
   // If ANY alarm is Disabled, Inhibited or Suppressed, set the Alarm Inhibit
   // summary status bit (which puts the "I" box on the graphic symbol).
   75: [XIC(FailToStart.Sts_AlmInh) ,XIC(FailToStop.Sts_AlmInh) ,XIC(IntlkTrip.Sts_AlmInh) ,XIC(DriveFault.Sts_AlmInh) ,XIC(IOFault.Sts_AlmInh) ]OTE(Sts_AlmInh);
